gfCNCPoint5[26380] = {X 520.4681, Y 51.2791, Z -8.0000, A 0.000, B 0.000, C 0.000 }
gfCNCPoint5[26381] = {X 519.7998, Y 51.2791, Z -8.0000, A 0.000, B 0.000, C 0.000 }
gfCNCPoint5[26382] = {X 518.8207, Y 51.1688, Z -8.0000, A 0.000, B 0.000, C 0.000 }
gfCNCPoint5[26383] = {X 517.8907, Y 50.8434, Z -8.0000, A 0.000, B 0.000, C 0.000 }
gfCNCPoint5[26384] = {X 517.0564, Y 50.3192, Z -8.0000, A 0.000, B 0.000, C 0.000 }
gfCNCPoint5[26385] = {X 516.3597, Y 49.6225, Z -8.0000, A 0.000, B 0.000, C 0.000 }
gfCNCPoint5[26386] = {X 515.8355, Y 48.7882, Z -8.0000, A 0.000, B 0.000, C 0.000 }
gfCNCPoint5[26387] = {X 515.5101, Y 47.8582, Z -8.0000, A 0.000, B 0.000, C 0.000 }
gfCNCPoint5[26388] = {X 515.3998, Y 46.8791, Z -8.0000, A 0.000, B 0.000, C 0.000 }
gfCNCPoint5[26389] = {X 515.3998, Y 39.9011, Z -8.0000, A 0.000, B 0.000, C 0.000 }
gfCNCPoint5[26390] = {X 515.5101, Y 38.9220, Z -8.0000, A 0.000, B 0.000, C 0.000 }
gfCNCPoint5[26391] = {X 515.8355, Y 37.9920, Z -8.0000, A 0.000, B 0.000, C 0.000 }
gfCNCPoint5[26392] = {X 516.3597, Y 37.1577, Z -8.0000, A 0.000, B 0.000, C 0.000 }
gfCNCPoint5[26393] = {X 517.0564, Y 36.4610, Z -8.0000, A 0.000, B 0.000, C 0.000 }
gfCNCPoint5[26394] = {X 517.8907, Y 35.9368, Z -8.0000, A 0.000, B 0.000, C 0.000 }
gfCNCPoint5[26395] = {X 518.8207, Y 35.6114, Z -8.0000, A 0.000, B 0.000, C 0.000 }
gfCNCPoint5[26396] = {X 519.7998, Y 35.5011, Z -8.0000, A 0.000, B 0.000, C 0.000 }
gfCNCPoint5[26397] = {X 520.5280, Y 35.5015, Z -8.0000, A 0.000, B 0.000, C 0.000 }
gfCNCPoint5[26398] = {X 521.3612, Y 35.5927, Z -8.0000, A 0.000, B 0.000, C 0.000 }
gfCNCPoint5[26399] = {X 522.1620, Y 35.8402, Z -8.0000, A 0.000, B 0.000, C 0.000 }
gfCNCPoint5[26400] = {X 522.9013, Y 36.2351, Z -8.0000, A 0.000, B 0.000, C 0.000 }
gfCNCPoint5[26401] = {X 523.5524, Y 36.7630, Z -8.0000, A 0.000, B 0.000, C 0.000 }
gfCNCPoint5[26402] = {X 524.0915, Y 37.4048, Z -8.0000, A 0.000, B 0.000, C 0.000 }
gfCNCPoint5[26403] = {X 534.5519, Y 37.4048, Z -8.0000, A 0.000, B 0.000, C 0.000 }
gfCNCPoint5[26404] = {X 534.5519, Y 34.0464, Z -8.0000, A 0.000, B 0.000, C 0.000 }
gfCNCPoint5[26405] = {X 530.1514, Y 34.0463, Z -8.0000, A 0.000, B 0.000, C 0.000 }
gfCNCPoint5[26406] = {X 529.6037, Y 34.6963, Z -8.0000, A 0.000, B 0.000, C 0.000 }
gfCNCPoint5[26407] = {X 528.9413, Y 35.2289, Z -8.0000, A 0.000, B 0.000, C 0.000 }
gfCNCPoint5[26408] = {X 528.1888, Y 35.6242, Z -8.0000, A 0.000, B 0.000, C 0.000 }
gfCNCPoint5[26409] = {X 527.3744, Y 35.8674, Z -8.0000, A 0.000, B 0.000, C 0.000 }
gfCNCPoint5[26410] = {X 526.5283, Y 35.9495, Z -8.0000, A 0.000, B 0.000, C 0.000 }
gfCNCPoint5[26411] = {X 525.8868, Y 35.9495, Z -8.0000, A 0.000, B 0.000, C 0.000 }
gfCNCPoint5[26412] = {X 524.9077, Y 35.8391, Z -8.0000, A 0.000, B 0.000, C 0.000 }
gfCNCPoint5[26413] = {X 523.9777, Y 35.5137, Z -8.0000, A 0.000, B 0.000, C 0.000 }
gfCNCPoint5[26414] = {X 523.1434, Y 34.9895, Z -8.0000, A 0.000, B 0.000, C 0.000 }
gfCNCPoint5[26415] = {X 522.4467, Y 34.2928, Z -8.0000, A 0.000, B 0.000, C 0.000 }
gfCNCPoint5[26416] = {X 521.9225, Y 33.4585, Z -8.0000, A 0.000, B 0.000, C 0.000 }
gfCNCPoint5[26417] = {X 521.5971, Y 32.5285, Z -8.0000, A 0.000, B 0.000, C 0.000 }
gfCNCPoint5[26418] = {X 521.4868, Y 31.5495, Z -8.0000, A 0.000, B 0.000, C 0.000 }
gfCNCPoint5[26419] = {X 521.4868, Y 24.5714, Z -8.0000, A 0.000, B 0.000, C 0.000 }
gfCNCPoint5[26420] = {X 521.5971, Y 23.5923, Z -8.0000, A 0.000, B 0.000, C 0.000 }
gfCNCPoint5[26421] = {X 521.9225, Y 22.6623, Z -8.0000, A 0.000, B 0.000, C 0.000 }
gfCNCPoint5[26422] = {X 522.4467, Y 21.8281, Z -8.0000, A 0.000, B 0.000, C 0.000 }
gfCNCPoint5[26423] = {X 523.1434, Y 21.1314, Z -8.0000, A 0.000, B 0.000, C 0.000 }
gfCNCPoint5[26424] = {X 523.9777, Y 20.6072, Z -8.0000, A 0.000, B 0.000, C 0.000 }
gfCNCPoint5[26425] = {X 524.9077, Y 20.2817, Z -8.0000, A 0.000, B 0.000, C 0.000 }
gfCNCPoint5[26426] = {X 525.8868, Y 20.1714, Z -8.0000, A 0.000, B 0.000, C 0.000 }
gfCNCPoint5[26427] = {X 526.5702, Y 20.1716, Z -8.0000, A 0.000, B 0.000, C 0.000 }
gfCNCPoint5[26428] = {X 527.4020, Y 20.2590, Z -8.0000, A 0.000, B 0.000, C 0.000 }
gfCNCPoint5[26429] = {X 528.2022, Y 20.5022, Z -8.0000, A 0.000, B 0.000, C 0.000 }
gfCNCPoint5[26430] = {X 528.9419, Y 20.8924, Z -8.0000, A 0.000, B 0.000, C 0.000 }
gfCNCPoint5[26431] = {X 529.5945, Y 21.4156, Z -8.0000, A 0.000, B 0.000, C 0.000 }
gfCNCPoint5[26432] = {X 530.1362, Y 22.0527, Z -8.0000, A 0.000, B 0.000, C 0.000 }
gfCNCPoint5[26433] = {X 534.5519, Y 22.0527, Z -8.0000, A 0.000, B 0.000, C 0.000 }
gfCNCPoint5[26434] = {X 534.5519, Y 19.7828, Z -8.0000, A 0.000, B 0.000, C 0.000 }
gfCNCPoint5[26435] = {X 528.8197, Y 19.7828, Z -8.0000, A 0.000, B 0.000, C 0.000 }
gfCNCPoint5[26436] = {X 528.8197, Y 20.2628, Z -8.0000, A 0.000, B 0.000, C 0.000 }
gfCNCPoint5[26437] = {X 534.0719, Y 20.2628, Z -8.0000, A 0.000, B 0.000, C 0.000 }
gfCNCPoint5[26438] = {X 534.0719, Y 21.5727, Z -8.0000, A 0.000, B 0.000, C 0.000 }
gfCNCPoint5[26439] = {X 530.3784, Y 21.5727, Z -8.0000, A 0.000, B 0.000, C 0.000 }
gfCNCPoint5[26440] = {X 529.6681, Y 20.8356, Z -8.0000, A 0.000, B 0.000, C 0.000 }
gfCNCPoint5[26441] = {X 528.8197, Y 20.2628, Z -8.0000, A 0.000, B 0.000, C 0.000 }
gfCNCPoint5[26442] = {X 528.8197, Y 19.7828, Z -8.0000, A 0.000, B 0.000, C 0.000 }
gfCNCPoint5[26443] = {X 524.2336, Y 19.7828, Z -8.0000, A 0.000, B 0.000, C 0.000 }
gfCNCPoint5[26444] = {X 523.6859, Y 20.4327, Z -8.0000, A 0.000, B 0.000, C 0.000 }
gfCNCPoint5[26445] = {X 523.0235, Y 20.9652, Z -8.0000, A 0.000, B 0.000, C 0.000 }
gfCNCPoint5[26446] = {X 522.2711, Y 21.3604, Z -8.0000, A 0.000, B 0.000, C 0.000 }
gfCNCPoint5[26447] = {X 521.4567, Y 21.6036, Z -8.0000, A 0.000, B 0.000, C 0.000 }
gfCNCPoint5[26448] = {X 520.6107, Y 21.6857, Z -8.0000, A 0.000, B 0.000, C 0.000 }
gfCNCPoint5[26449] = {X 519.9691, Y 21.6857, Z -8.0000, A 0.000, B 0.000, C 0.000 }
gfCNCPoint5[26450] = {X 518.9900, Y 21.5754, Z -8.0000, A 0.000, B 0.000, C 0.000 }
gfCNCPoint5[26451] = {X 518.0600, Y 21.2500, Z -8.0000, A 0.000, B 0.000, C 0.000 }
gfCNCPoint5[26452] = {X 517.2257, Y 20.7258, Z -8.0000, A 0.000, B 0.000, C 0.000 }
gfCNCPoint5[26453] = {X 516.5290, Y 20.0291, Z -8.0000, A 0.000, B 0.000, C 0.000 }
gfCNCPoint5[26454] = {X 516.0048, Y 19.1948, Z -8.0000, A 0.000, B 0.000, C 0.000 }
gfCNCPoint5[26455] = {X 515.6794, Y 18.2648, Z -8.0000, A 0.000, B 0.000, C 0.000 }
gfCNCPoint5[26456] = {X 515.5691, Y 17.2857, Z -8.0000, A 0.000, B 0.000, C 0.000 }
gfCNCPoint5[26457] = {X 515.5691, Y 10.3077, Z -8.0000, A 0.000, B 0.000, C 0.000 }
gfCNCPoint5[26458] = {X 515.6394, Y 9.5244, Z -8.0000, A 0.000, B 0.000, C 0.000 }
gfCNCPoint5[26459] = {X 515.8480, Y 8.7661, Z -8.0000, A 0.000, B 0.000, C 0.000 }
gfCNCPoint5[26460] = {X 516.1883, Y 8.0570, Z -8.0000, A 0.000, B 0.000, C 0.000 }
gfCNCPoint5[26461] = {X 516.6494, Y 7.4199, Z -8.0000, A 0.000, B 0.000, C 0.000 }
gfCNCPoint5[26462] = {X 516.2873, Y 7.1048, Z -8.0000, A 0.000, B 0.000, C 0.000 }
gfCNCPoint5[26463] = {X 370.1008, Y 7.1048, Z -8.0000, A 0.000, B 0.000, C 0.000 }
gfCNCPoint5[26464] = {X 371.1247, Y 8.7921, Z -8.0000, A 0.000, B 0.000, C 0.000 }
gfCNCPoint5[26465] = {X 372.0360, Y 10.5428, Z -8.0000, A 0.000, B 0.000, C 0.000 }
gfCNCPoint5[26466] = {X 372.8329, Y 12.3542, Z -8.0000, A 0.000, B 0.000, C 0.000 }
gfCNCPoint5[26467] = {X 373.5091, Y 14.2140, Z -8.0000, A 0.000, B 0.000, C 0.000 }
gfCNCPoint5[26468] = {X 374.0619, Y 16.1141, Z -8.0000, A 0.000, B 0.000, C 0.000 }
gfCNCPoint5[26469] = {X 374.6092, Y 18.6904, Z -8.0000, A 0.000, B 0.000, C 0.000 }
gfCNCPoint5[26470] = {X 374.9714, Y 21.2992, Z -8.0000, A 0.000, B 0.000, C 0.000 }
gfCNCPoint5[26471] = {X 375.1469, Y 23.9271, Z -8.0000, A 0.000, B 0.000, C 0.000 }
gfCNCPoint5[26472] = {X 375.1347, Y 26.5608, Z -8.0000, A 0.000, B 0.000, C 0.000 }
gfCNCPoint5[26473] = {X 374.9349, Y 29.1870, Z -8.0000, A 0.000, B 0.000, C 0.000 }
gfCNCPoint5[26474] = {X 374.5485, Y 31.7923, Z -8.0000, A 0.000, B 0.000, C 0.000 }
gfCNCPoint5[26475] = {X 386.3483, Y 33.9749, Z -8.0000, A 0.000, B 0.000, C 0.000 }
gfCNCPoint5[26476] = {X 386.2676, Y 34.4005, Z -8.0000, A 0.000, B 0.000, C 0.000 }
gfCNCPoint5[26477] = {X 386.1832, Y 34.8254, Z -8.0000, A 0.000, B 0.000, C 0.000 }
gfCNCPoint5[26478] = {X 386.0243, Y 35.5742, Z -8.0000, A 0.000, B 0.000, C 0.000 }
gfCNCPoint5[26479] = {X 385.8518, Y 36.3200, Z -8.0000, A 0.000, B 0.000, C 0.000 }
gfCNCPoint5[26480] = {X 386.9552, Y 36.3200, Z -8.0000, A 0.000, B 0.000, C 0.000 }
gfCNCPoint5[26481] = {X 386.9552, Y 35.0303, Z -8.0000, A 0.000, B 0.000, C 0.000 }
gfCNCPoint5[26482] = {X 386.3483, Y 33.9749, Z -8.0000, A 0.000, B 0.000, C 0.000 }
gfCNCPoint5[26483] = {X 383.9884, Y 33.5384, Z -8.0000, A 0.000, B 0.000, C 0.000 }
gfCNCPoint5[26484] = {X 383.9116, Y 33.9435, Z -8.0000, A 0.000, B 0.000, C 0.000 }
gfCNCPoint5[26485] = {X 383.8312, Y 34.3479, Z -8.0000, A 0.000, B 0.000, C 0.000 }
gfCNCPoint5[26486] = {X 383.6813, Y 35.0543, Z -8.0000, A 0.000, B 0.000, C 0.000 }
gfCNCPoint5[26487] = {X 383.5186, Y 35.7577, Z -8.0000, A 0.000, B 0.000, C 0.000 }
gfCNCPoint5[26488] = {X 383.1288, Y 37.2470, Z -8.0000, A 0.000, B 0.000, C 0.000 }
gfCNCPoint5[26489] = {X 382.6813, Y 38.7200, Z -8.0000, A 0.000, B 0.000, C 0.000 }
gfCNCPoint5[26490] = {X 388.0597, Y 38.7200, Z -8.0000, A 0.000, B 0.000, C 0.000 }
gfCNCPoint5[26491] = {X 388.4821, Y 38.7246, Z -8.0000, A 0.000, B 0.000, C 0.000 }
gfCNCPoint5[26492] = {X 388.9043, Y 38.7385, Z -8.0000, A 0.000, B 0.000, C 0.000 }
gfCNCPoint5[26493] = {X 389.1204, Y 38.2363, Z -8.0000, A 0.000, B 0.000, C 0.000 }
gfCNCPoint5[26494] = {X 389.3552, Y 37.7427, Z -8.0000, A 0.000, B 0.000, C 0.000 }
gfCNCPoint5[26495] = {X 389.3552, Y 34.3894, Z -8.0000, A 0.000, B 0.000, C 0.000 }
gfCNCPoint5[26496] = {X 384.7465, Y 26.3749, Z -8.0000, A 0.000, B 0.000, C 0.000 }
gfCNCPoint5[26497] = {X 384.6173, Y 28.7747, Z -8.0000, A 0.000, B 0.000, C 0.000 }
gfCNCPoint5[26498] = {X 384.3643, Y 31.1647, Z -8.0000, A 0.000, B 0.000, C 0.000 }
gfCNCPoint5[26499] = {X 383.9884, Y 33.5384, Z -8.0000, A 0.000, B 0.000, C 0.000 }
gfCNCPoint5[26500] = {X 381.6284, Y 33.1019, Z -8.0000, A 0.000, B 0.000, C 0.000 }
gfCNCPoint5[26501] = {X 381.5555, Y 33.4865, Z -8.0000, A 0.000, B 0.000, C 0.000 }
gfCNCPoint5[26502] = {X 381.4792, Y 33.8705, Z -8.0000, A 0.000, B 0.000, C 0.000 }
gfCNCPoint5[26503] = {X 380.9979, Y 35.9396, Z -8.0000, A 0.000, B 0.000, C 0.000 }
gfCNCPoint5[26504] = {X 380.3990, Y 37.9777, Z -8.0000, A 0.000, B 0.000, C 0.000 }
gfCNCPoint5[26505] = {X 379.8437, Y 39.5622, Z -8.0000, A 0.000, B 0.000, C 0.000 }
gfCNCPoint5[26506] = {X 379.2173, Y 41.1200, Z -8.0000, A 0.000, B 0.000, C 0.000 }
gfCNCPoint5[26507] = {X 388.0597, Y 41.1200, Z -8.0000, A 0.000, B 0.000, C 0.000 }
gfCNCPoint5[26508] = {X 389.3256, Y 41.1675, Z -8.0000, A 0.000, B 0.000, C 0.000 }
gfCNCPoint5[26509] = {X 390.5844, Y 41.3099, Z -8.0000, A 0.000, B 0.000, C 0.000 }
gfCNCPoint5[26510] = {X 391.0709, Y 39.7838, Z -8.0000, A 0.000, B 0.000, C 0.000 }
gfCNCPoint5[26511] = {X 391.7552, Y 38.3355, Z -8.0000, A 0.000, B 0.000, C 0.000 }
gfCNCPoint5[26512] = {X 391.7552, Y 33.7486, Z -8.0000, A 0.000, B 0.000, C 0.000 }
gfCNCPoint5[26513] = {X 386.7075, Y 24.9707, Z -8.0000, A 0.000, B 0.000, C 0.000 }
gfCNCPoint5[26514] = {X 386.1105, Y 23.9508, Z -8.0000, A 0.000, B 0.000, C 0.000 }
gfCNCPoint5[26515] = {X 385.4975, Y 22.9404, Z -8.0000, A 0.000, B 0.000, C 0.000 }
gfCNCPoint5[26516] = {X 384.4699, Y 22.1514, Z -8.0000, A 0.000, B 0.000, C 0.000 }
gfCNCPoint5[26517] = {X 383.5327, Y 21.2569, Z -8.0000, A 0.000, B 0.000, C 0.000 }
gfCNCPoint5[26518] = {X 382.6966, Y 20.2672, Z -8.0000, A 0.000, B 0.000, C 0.000 }
gfCNCPoint5[26519] = {X 381.9714, Y 19.1936, Z -8.0000, A 0.000, B 0.000, C 0.000 }
gfCNCPoint5[26520] = {X 382.2245, Y 21.5571, Z -8.0000, A 0.000, B 0.000, C 0.000 }
gfCNCPoint5[26521] = {X 382.3499, Y 23.9308, Z -8.0000, A 0.000, B 0.000, C 0.000 }
gfCNCPoint5[26522] = {X 382.3474, Y 26.3077, Z -8.0000, A 0.000, B 0.000, C 0.000 }
gfCNCPoint5[26523] = {X 382.2249, Y 28.5838, Z -8.0000, A 0.000, B 0.000, C 0.000 }
gfCNCPoint5[26524] = {X 381.9850, Y 30.8506, Z -8.0000, A 0.000, B 0.000, C 0.000 }
gfCNCPoint5[26525] = {X 381.6284, Y 33.1019, Z -8.0000, A 0.000, B 0.000, C 0.000 }
gfCNCPoint5[26526] = {X 379.2684, Y 32.6654, Z -8.0000, A 0.000, B 0.000, C 0.000 }
gfCNCPoint5[26527] = {X 379.1994, Y 33.0295, Z -8.0000, A 0.000, B 0.000, C 0.000 }
gfCNCPoint5[26528] = {X 379.1271, Y 33.3931, Z -8.0000, A 0.000, B 0.000, C 0.000 }
gfCNCPoint5[26529] = {X 378.5771, Y 35.7000, Z -8.0000, A 0.000, B 0.000, C 0.000 }
gfCNCPoint5[26530] = {X 377.8708, Y 37.9640, Z -8.0000, A 0.000, B 0.000, C 0.000 }
gfCNCPoint5[26531] = {X 377.0114, Y 40.1744, Z -8.0000, A 0.000, B 0.000, C 0.000 }
gfCNCPoint5[26532] = {X 376.2302, Y 41.8694, Z -8.0000, A 0.000, B 0.000, C 0.000 }
gfCNCPoint5[26533] = {X 375.3590, Y 43.5200, Z -8.0000, A 0.000, B 0.000, C 0.000 }
gfCNCPoint5[26534] = {X 388.0597, Y 43.5200, Z -8.0000, A 0.000, B 0.000, C 0.000 }
gfCNCPoint5[26535] = {X 389.6072, Y 43.6029, Z -8.0000, A 0.000, B 0.000, C 0.000 }
gfCNCPoint5[26536] = {X 391.1370, Y 43.8508, Z -8.0000, A 0.000, B 0.000, C 0.000 }
gfCNCPoint5[26537] = {X 392.6316, Y 44.2607, Z -8.0000, A 0.000, B 0.000, C 0.000 }
gfCNCPoint5[26538] = {X 392.7236, Y 42.8756, Z -8.0000, A 0.000, B 0.000, C 0.000 }
gfCNCPoint5[26539] = {X 393.0129, Y 41.5179, Z -8.0000, A 0.000, B 0.000, C 0.000 }
gfCNCPoint5[26540] = {X 393.4934, Y 40.2155, Z -8.0000, A 0.000, B 0.000, C 0.000 }
gfCNCPoint5[26541] = {X 394.1552, Y 38.9952, Z -8.0000, A 0.000, B 0.000, C 0.000 }
gfCNCPoint5[26542] = {X 394.1552, Y 33.1077, Z -8.0000, A 0.000, B 0.000, C 0.000 }
gfCNCPoint5[26543] = {X 388.7881, Y 23.7743, Z -8.0000, A 0.000, B 0.000, C 0.000 }
gfCNCPoint5[26544] = {X 388.0333, Y 22.4902, Z -8.0000, A 0.000, B 0.000, C 0.000 }
gfCNCPoint5[26545] = {X 387.2543, Y 21.2208, Z -8.0000, A 0.000, B 0.000, C 0.000 }
gfCNCPoint5[26546] = {X 386.3070, Y 20.5563, Z -8.0000, A 0.000, B 0.000, C 0.000 }
gfCNCPoint5[26547] = {X 385.4458, Y 19.7835, Z -8.0000, A 0.000, B 0.000, C 0.000 }
gfCNCPoint5[26548] = {X 384.6829, Y 18.9135, Z -8.0000, A 0.000, B 0.000, C 0.000 }
gfCNCPoint5[26549] = {X 384.0293, Y 17.9587, Z -8.0000, A 0.000, B 0.000, C 0.000 }
gfCNCPoint5[26550] = {X 383.4406, Y 16.8105, Z -8.0000, A 0.000, B 0.000, C 0.000 }
gfCNCPoint5[26551] = {X 383.0098, Y 15.5941, Z -8.0000, A 0.000, B 0.000, C 0.000 }
gfCNCPoint5[26552] = {X 382.7447, Y 14.3312, Z -8.0000, A 0.000, B 0.000, C 0.000 }
gfCNCPoint5[26553] = {X 382.6498, Y 13.0443, Z -8.0000, A 0.000, B 0.000, C 0.000 }
gfCNCPoint5[26554] = {X 382.6496, Y 12.1868, Z -8.0000, A 0.000, B 0.000, C 0.000 }
gfCNCPoint5[26555] = {X 382.6507, Y 12.0458, Z -8.0000, A 0.000, B 0.000, C 0.000 }
gfCNCPoint5[26556] = {X 382.6537, Y 11.9048, Z -8.0000, A 0.000, B 0.000, C 0.000 }
gfCNCPoint5[26557] = {X 377.7930, Y 11.9048, Z -8.0000, A 0.000, B 0.000, C 0.000 }
gfCNCPoint5[26558] = {X 378.2878, Y 13.4079, Z -8.0000, A 0.000, B 0.000, C 0.000 }
gfCNCPoint5[26559] = {X 378.7141, Y 14.9319, Z -8.0000, A 0.000, B 0.000, C 0.000 }
gfCNCPoint5[26560] = {X 379.2175, Y 17.2103, Z -8.0000, A 0.000, B 0.000, C 0.000 }
gfCNCPoint5[26561] = {X 379.5928, Y 19.5133, Z -8.0000, A 0.000, B 0.000, C 0.000 }
gfCNCPoint5[26562] = {X 379.8616, Y 22.1413, Z -8.0000, A 0.000, B 0.000, C 0.000 }
gfCNCPoint5[26563] = {X 379.9637, Y 24.7812, Z -8.0000, A 0.000, B 0.000, C 0.000 }
gfCNCPoint5[26564] = {X 379.8985, Y 27.4221, Z -8.0000, A 0.000, B 0.000, C 0.000 }
gfCNCPoint5[26565] = {X 379.6665, Y 30.0537, Z -8.0000, A 0.000, B 0.000, C 0.000 }
gfCNCPoint5[26566] = {X 379.2684, Y 32.6654, Z -8.0000, A 0.000, B 0.000, C 0.000 }
gfCNCPoint5[26567] = {X 376.9085, Y 32.2288, Z -8.0000, A 0.000, B 0.000, C 0.000 }
gfCNCPoint5[26568] = {X 376.8433, Y 32.5725, Z -8.0000, A 0.000, B 0.000, C 0.000 }
gfCNCPoint5[26569] = {X 376.7751, Y 32.9156, Z -8.0000, A 0.000, B 0.000, C 0.000 }
gfCNCPoint5[26570] = {X 376.1777, Y 35.3682, Z -8.0000, A 0.000, B 0.000, C 0.000 }
gfCNCPoint5[26571] = {X 375.3905, Y 37.7667, Z -8.0000, A 0.000, B 0.000, C 0.000 }
gfCNCPoint5[26572] = {X 374.4185, Y 40.0964, Z -8.0000, A 0.000, B 0.000, C 0.000 }
gfCNCPoint5[26573] = {X 373.2674, Y 42.3430, Z -8.0000, A 0.000, B 0.000, C 0.000 }
gfCNCPoint5[26574] = {X 372.1530, Y 44.1780, Z -8.0000, A 0.000, B 0.000, C 0.000 }
gfCNCPoint5[26575] = {X 370.9191, Y 45.9349, Z -8.0000, A 0.000, B 0.000, C 0.000 }
gfCNCPoint5[26576] = {X 371.2191, Y 45.9237, Z -8.0000, A 0.000, B 0.000, C 0.000 }
gfCNCPoint5[26577] = {X 371.5193, Y 45.9200, Z -8.0000, A 0.000, B 0.000, C 0.000 }
gfCNCPoint5[26578] = {X 388.0597, Y 45.9200, Z -8.0000, A 0.000, B 0.000, C 0.000 }
gfCNCPoint5[26579] = {X 389.4143, Y 45.9962, Z -8.0000, A 0.000, B 0.000, C 0.000 }
gfCNCPoint5[26580] = {X 390.7519, Y 46.2238, Z -8.0000, A 0.000, B 0.000, C 0.000 }
gfCNCPoint5[26581] = {X 392.0555, Y 46.6000, Z -8.0000, A 0.000, B 0.000, C 0.000 }
gfCNCPoint5[26582] = {X 393.3087, Y 47.1200, Z -8.0000, A 0.000, B 0.000, C 0.000 }
gfCNCPoint5[26583] = {X 394.2237, Y 46.7243, Z -8.0000, A 0.000, B 0.000, C 0.000 }
gfCNCPoint5[26584] = {X 395.1681, Y 46.4053, Z -8.0000, A 0.000, B 0.000, C 0.000 }
gfCNCPoint5[26585] = {X 395.0678, Y 45.7292, Z -8.0000, A 0.000, B 0.000, C 0.000 }
gfCNCPoint5[26586] = {X 395.0314, Y 45.0468, Z -8.0000, A 0.000, B 0.000, C 0.000 }
gfCNCPoint5[26587] = {X 395.0316, Y 44.1296, Z -8.0000, A 0.000, B 0.000, C 0.000 }
gfCNCPoint5[26588] = {X 395.1397, Y 42.9564, Z -8.0000, A 0.000, B 0.000, C 0.000 }
gfCNCPoint5[26589] = {X 395.4356, Y 41.8161, Z -8.0000, A 0.000, B 0.000, C 0.000 }
gfCNCPoint5[26590] = {X 395.9116, Y 40.7384, Z -8.0000, A 0.000, B 0.000, C 0.000 }
gfCNCPoint5[26591] = {X 396.5552, Y 39.7516, Z -8.0000, A 0.000, B 0.000, C 0.000 }
gfCNCPoint5[26592] = {X 396.5552, Y 32.4669, Z -8.0000, A 0.000, B 0.000, C 0.000 }
gfCNCPoint5[26593] = {X 390.8686, Y 22.5779, Z -8.0000, A 0.000, B 0.000, C 0.000 }
gfCNCPoint5[26594] = {X 390.0503, Y 21.1873, Z -8.0000, A 0.000, B 0.000, C 0.000 }
gfCNCPoint5[26595] = {X 389.2044, Y 19.8133, Z -8.0000, A 0.000, B 0.000, C 0.000 }
gfCNCPoint5[26596] = {X 389.0604, Y 19.6016, Z -8.0000, A 0.000, B 0.000, C 0.000 }
gfCNCPoint5[26597] = {X 388.9019, Y 19.4005, Z -8.0000, A 0.000, B 0.000, C 0.000 }
gfCNCPoint5[26598] = {X 387.8143, Y 18.6886, Z -8.0000, A 0.000, B 0.000, C 0.000 }
gfCNCPoint5[26599] = {X 386.8707, Y 17.7945, Z -8.0000, A 0.000, B 0.000, C 0.000 }
gfCNCPoint5[26600] = {X 386.1011, Y 16.7469, Z -8.0000, A 0.000, B 0.000, C 0.000 }
gfCNCPoint5[26601] = {X 385.5302, Y 15.5791, Z -8.0000, A 0.000, B 0.000, C 0.000 }
gfCNCPoint5[26602] = {X 385.1760, Y 14.3284, Z -8.0000, A 0.000, B 0.000, C 0.000 }
gfCNCPoint5[26603] = {X 385.0498, Y 13.0347, Z -8.0000, A 0.000, B 0.000, C 0.000 }
gfCNCPoint5[26604] = {X 385.0496, Y 12.1868, Z -8.0000, A 0.000, B 0.000, C 0.000 }
gfCNCPoint5[26605] = {X 385.0504, Y 12.0808, Z -8.0000, A 0.000, B 0.000, C 0.000 }
gfCNCPoint5[26606] = {X 385.0527, Y 11.9747, Z -8.0000, A 0.000, B 0.000, C 0.000 }
gfCNCPoint5[26607] = {X 385.1994, Y 10.7176, Z -8.0000, A 0.000, B 0.000, C 0.000 }
gfCNCPoint5[26608] = {X 385.5617, Y 9.5048, Z -8.0000, A 0.000, B 0.000, C 0.000 }
gfCNCPoint5[26609] = {X 374.2000, Y 9.5048, Z -8.0000, A 0.000, B 0.000, C 0.000 }
gfCNCPoint5[26610] = {X 374.9081, Y 11.0880, Z -8.0000, A 0.000, B 0.000, C 0.000 }
gfCNCPoint5[26611] = {X 375.5309, Y 12.7067, Z -8.0000, A 0.000, B 0.000, C 0.000 }
gfCNCPoint5[26612] = {X 375.9918, Y 14.1066, Z -8.0000, A 0.000, B 0.000, C 0.000 }
gfCNCPoint5[26613] = {X 376.3888, Y 15.5259, Z -8.0000, A 0.000, B 0.000, C 0.000 }
gfCNCPoint5[26614] = {X 376.9722, Y 18.2705, Z -8.0000, A 0.000, B 0.000, C 0.000 }
gfCNCPoint5[26615] = {X 377.3585, Y 21.0497, Z -8.0000, A 0.000, B 0.000, C 0.000 }
gfCNCPoint5[26616] = {X 377.5457, Y 23.8494, Z -8.0000, A 0.000, B 0.000, C 0.000 }
gfCNCPoint5[26617] = {X 377.5329, Y 26.6554, Z -8.0000, A 0.000, B 0.000, C 0.000 }
gfCNCPoint5[26618] = {X 377.3201, Y 29.4532, Z -8.0000, A 0.000, B 0.000, C 0.000 }
gfCNCPoint5[26619] = {X 376.9085, Y 32.2288, Z -8.0000, A 0.000, B 0.000, C 0.000 }
gfCNCPoint5[26620] = {X 374.5485, Y 31.7923, Z -8.0000, A 0.000, B 0.000, C 0.000 }
gfCNCPoint5[26621] = {X 374.4872, Y 32.1155, Z -8.0000, A 0.000, B 0.000, C 0.000 }
gfCNCPoint5[26622] = {X 374.4231, Y 32.4381, Z -8.0000, A 0.000, B 0.000, C 0.000 }
gfCNCPoint5[26623] = {X 373.8982, Y 34.6095, Z -8.0000, A 0.000, B 0.000, C 0.000 }
gfCNCPoint5[26624] = {X 373.2127, Y 36.7356, Z -8.0000, A 0.000, B 0.000, C 0.000 }
gfCNCPoint5[26625] = {X 372.3703, Y 38.8046, Z -8.0000, A 0.000, B 0.000, C 0.000 }
gfCNCPoint5[26626] = {X 371.3758, Y 40.8049, Z -8.0000, A 0.000, B 0.000, C 0.000 }
gfCNCPoint5[26627] = {X 370.2347, Y 42.7254, Z -8.0000, A 0.000, B 0.000, C 0.000 }
gfCNCPoint5[26628] = {X 368.9534, Y 44.5554, Z -8.0000, A 0.000, B 0.000, C 0.000 }
gfCNCPoint5[26629] = {X 367.5572, Y 46.2628, Z -8.0000, A 0.000, B 0.000, C 0.000 }
gfCNCPoint5[26630] = {X 366.0280, Y 47.8522, Z -8.0000, A 0.000, B 0.000, C 0.000 }
gfCNCPoint5[26631] = {X 364.3756, Y 49.3132, Z -8.0000, A 0.000, B 0.000, C 0.000 }
gfCNCPoint5[26632] = {X 362.6108, Y 50.6362, Z -8.0000, A 0.000, B 0.000, C 0.000 }
gfCNCPoint5[26633] = {X 360.7452, Y 51.8127, Z -8.0000, A 0.000, B 0.000, C 0.000 }
gfCNCPoint5[26634] = {X 358.7908, Y 52.8350, Z -8.0000, A 0.000, B 0.000, C 0.000 }
gfCNCPoint5[26635] = {X 358.6057, Y 52.9216, Z -8.0000, A 0.000, B 0.000, C 0.000 }
gfCNCPoint5[26636] = {X 358.4200, Y 53.0069, Z -8.0000, A 0.000, B 0.000, C 0.000 }
gfCNCPoint5[26637] = {X 356.1467, Y 53.8835, Z -8.0000, A 0.000, B 0.000, C 0.000 }
gfCNCPoint5[26638] = {X 353.8065, Y 54.5619, Z -8.0000, A 0.000, B 0.000, C 0.000 }
gfCNCPoint5[26639] = {X 351.4168, Y 55.0371, Z -8.0000, A 0.000, B 0.000, C 0.000 }
gfCNCPoint5[26640] = {X 348.9952, Y 55.3056, Z -8.0000, A 0.000, B 0.000, C 0.000 }
gfCNCPoint5[26641] = {X 349.9664, Y 69.6728, Z -8.0000, A 0.000, B 0.000, C 0.000 }
gfCNCPoint5[26642] = {X 348.6648, Y 69.7409, Z -8.0000, A 0.000, B 0.000, C 0.000 }
gfCNCPoint5[26643] = {X 347.3618, Y 69.7693, Z -8.0000, A 0.000, B 0.000, C 0.000 }
gfCNCPoint5[26644] = {X 346.5844, Y 69.7785, Z -8.0000, A 0.000, B 0.000, C 0.000 }
gfCNCPoint5[26645] = {X 345.8070, Y 69.7737, Z -8.0000, A 0.000, B 0.000, C 0.000 }
gfCNCPoint5[26646] = {X 345.5918, Y 70.1904, Z -8.0000, A 0.000, B 0.000, C 0.000 }
gfCNCPoint5[26647] = {X 345.3684, Y 70.6028, Z -8.0000, A 0.000, B 0.000, C 0.000 }
gfCNCPoint5[26648] = {X 347.2082, Y 70.6201, Z -8.0000, A 0.000, B 0.000, C 0.000 }
gfCNCPoint5[26649] = {X 349.0480, Y 70.6084, Z -8.0000, A 0.000, B 0.000, C 0.000 }
gfCNCPoint5[26650] = {X 349.7516, Y 70.6081, Z -8.0000, A 0.000, B 0.000, C 0.000 }
gfCNCPoint5[26651] = {X 350.4553, Y 70.6025, Z -8.0000, A 0.000, B 0.000, C 0.000 }
gfCNCPoint5[26652] = {X 350.2058, Y 70.1403, Z -8.0000, A 0.000, B 0.000, C 0.000 }
gfCNCPoint5[26653] = {X 349.9664, Y 69.6728, Z -8.0000, A 0.000, B 0.000, C 0.000 }
gfCNCPoint5[26654] = {X 349.8045, Y 67.2783, Z -8.0000, A 0.000, B 0.000, C 0.000 }
gfCNCPoint5[26655] = {X 348.5675, Y 67.3429, Z -8.0000, A 0.000, B 0.000, C 0.000 }
gfCNCPoint5[26656] = {X 347.3291, Y 67.3695, Z -8.0000, A 0.000, B 0.000, C 0.000 }
gfCNCPoint5[26657] = {X 345.8126, Y 67.3735, Z -8.0000, A 0.000, B 0.000, C 0.000 }
gfCNCPoint5[26658] = {X 344.2969, Y 67.3217, Z -8.0000, A 0.000, B 0.000, C 0.000 }
gfCNCPoint5[26659] = {X 343.8118, Y 68.3945, Z -8.0000, A 0.000, B 0.000, C 0.000 }
gfCNCPoint5[26660] = {X 343.2692, Y 69.4395, Z -8.0000, A 0.000, B 0.000, C 0.000 }
gfCNCPoint5[26661] = {X 342.7891, Y 70.2628, Z -8.0000, A 0.000, B 0.000, C 0.000 }
gfCNCPoint5[26662] = {X 342.2734, Y 71.0641, Z -8.0000, A 0.000, B 0.000, C 0.000 }
gfCNCPoint5[26663] = {X 342.2736, Y 72.9104, Z -8.0000, A 0.000, B 0.000, C 0.000 }
gfCNCPoint5[26664] = {X 343.8000, Y 72.9662, Z -8.0000, A 0.000, B 0.000, C 0.000 }
gfCNCPoint5[26665] = {X 345.3269, Y 73.0024, Z -8.0000, A 0.000, B 0.000, C 0.000 }
gfCNCPoint5[26666] = {X 347.1940, Y 73.0201, Z -8.0000, A 0.000, B 0.000, C 0.000 }
gfCNCPoint5[26667] = {X 349.0612, Y 73.0085, Z -8.0000, A 0.000, B 0.000, C 0.000 }
gfCNCPoint5[26668] = {X 349.7722, Y 73.0080, Z -8.0000, A 0.000, B 0.000, C 0.000 }
gfCNCPoint5[26669] = {X 350.4831, Y 73.0024, Z -8.0000, A 0.000, B 0.000, C 0.000 }
gfCNCPoint5[26670] = {X 352.0210, Y 72.9723, Z -8.0000, A 0.000, B 0.000, C 0.000 }
gfCNCPoint5[26671] = {X 353.5582, Y 72.9179, Z -8.0000, A 0.000, B 0.000, C 0.000 }
gfCNCPoint5[26672] = {X 353.5581, Y 71.0756, Z -8.0000, A 0.000, B 0.000, C 0.000 }
gfCNCPoint5[26673] = {X 353.0382, Y 70.2687, Z -8.0000, A 0.000, B 0.000, C 0.000 }
gfCNCPoint5[26674] = {X 352.5547, Y 69.4396, Z -8.0000, A 0.000, B 0.000, C 0.000 }
gfCNCPoint5[26675] = {X 351.9680, Y 68.3027, Z -8.0000, A 0.000, B 0.000, C 0.000 }
gfCNCPoint5[26676] = {X 351.4495, Y 67.1332, Z -8.0000, A 0.000, B 0.000, C 0.000 }
gfCNCPoint5[26677] = {X 350.6278, Y 67.2142, Z -8.0000, A 0.000, B 0.000, C 0.000 }
gfCNCPoint5[26678] = {X 349.8045, Y 67.2783, Z -8.0000, A 0.000, B 0.000, C 0.000 }
gfCNCPoint5[26679] = {X 349.6427, Y 64.8838, Z -8.0000, A 0.000, B 0.000, C 0.000 }
gfCNCPoint5[26680] = {X 348.4702, Y 64.9448, Z -8.0000, A 0.000, B 0.000, C 0.000 }
gfCNCPoint5[26681] = {X 347.2964, Y 64.9696, Z -8.0000, A 0.000, B 0.000, C 0.000 }
gfCNCPoint5[26682] = {X 344.9826, Y 64.9504, Z -8.0000, A 0.000, B 0.000, C 0.000 }
gfCNCPoint5[26683] = {X 342.6741, Y 64.7932, Z -8.0000, A 0.000, B 0.000, C 0.000 }
gfCNCPoint5[26684] = {X 341.9396, Y 66.7276, Z -8.0000, A 0.000, B 0.000, C 0.000 }
gfCNCPoint5[26685] = {X 341.0024, Y 68.5724, Z -8.0000, A 0.000, B 0.000, C 0.000 }
gfCNCPoint5[26686] = {X 339.8733, Y 70.3064, Z -8.0000, A 0.000, B 0.000, C 0.000 }
gfCNCPoint5[26687] = {X 339.8738, Y 75.1877, Z -8.0000, A 0.000, B 0.000, C 0.000 }
gfCNCPoint5[26688] = {X 344.4720, Y 75.3853, Z -8.0000, A 0.000, B 0.000, C 0.000 }
gfCNCPoint5[26689] = {X 349.0745, Y 75.4085, Z -8.0000, A 0.000, B 0.000, C 0.000 }
gfCNCPoint5[26690] = {X 352.5183, Y 75.3586, Z -8.0000, A 0.000, B 0.000, C 0.000 }
gfCNCPoint5[26691] = {X 355.9583, Y 75.1895, Z -8.0000, A 0.000, B 0.000, C 0.000 }
gfCNCPoint5[26692] = {X 355.9580, Y 70.3167, Z -8.0000, A 0.000, B 0.000, C 0.000 }
gfCNCPoint5[26693] = {X 355.0507, Y 68.9593, Z -8.0000, A 0.000, B 0.000, C 0.000 }
gfCNCPoint5[26694] = {X 354.2615, Y 67.5299, Z -8.0000, A 0.000, B 0.000, C 0.000 }
gfCNCPoint5[26695] = {X 353.5961, Y 66.0388, Z -8.0000, A 0.000, B 0.000, C 0.000 }
gfCNCPoint5[26696] = {X 353.0592, Y 64.4968, Z -8.0000, A 0.000, B 0.000, C 0.000 }
gfCNCPoint5[26697] = {X 351.3553, Y 64.7290, Z -8.0000, A 0.000, B 0.000, C 0.000 }
gfCNCPoint5[26698] = {X 349.6427, Y 64.8838, Z -8.0000, A 0.000, B 0.000, C 0.000 }
gfCNCPoint5[26699] = {X 349.4808, Y 62.4892, Z -8.0000, A 0.000, B 0.000, C 0.000 }
gfCNCPoint5[26700] = {X 348.3729, Y 62.5468, Z -8.0000, A 0.000, B 0.000, C 0.000 }
gfCNCPoint5[26701] = {X 347.2638, Y 62.5698, Z -8.0000, A 0.000, B 0.000, C 0.000 }
gfCNCPoint5[26702] = {X 345.1284, Y 62.5542, Z -8.0000, A 0.000, B 0.000, C 0.000 }
gfCNCPoint5[26703] = {X 342.9976, Y 62.4133, Z -8.0000, A 0.000, B 0.000, C 0.000 }
gfCNCPoint5[26704] = {X 340.8787, Y 62.1476, Z -8.0000, A 0.000, B 0.000, C 0.000 }
gfCNCPoint5[26705] = {X 340.4890, Y 63.7352, Z -8.0000, A 0.000, B 0.000, C 0.000 }
gfCNCPoint5[26706] = {X 339.9479, Y 65.2779, Z -8.0000, A 0.000, B 0.000, C 0.000 }
gfCNCPoint5[26707] = {X 339.2604, Y 66.7611, Z -8.0000, A 0.000, B 0.000, C 0.000 }
gfCNCPoint5[26708] = {X 338.4329, Y 68.1710, Z -8.0000, A 0.000, B 0.000, C 0.000 }
gfCNCPoint5[26709] = {X 337.4732, Y 69.4944, Z -8.0000, A 0.000, B 0.000, C 0.000 }
gfCNCPoint5[26710] = {X 337.4740, Y 77.4231, Z -8.0000, A 0.000, B 0.000, C 0.000 }
gfCNCPoint5[26711] = {X 341.3406, Y 77.6726, Z -8.0000, A 0.000, B 0.000, C 0.000 }
gfCNCPoint5[26712] = {X 345.2131, Y 77.8012, Z -8.0000, A 0.000, B 0.000, C 0.000 }
gfCNCPoint5[26713] = {X 349.0878, Y 77.8086, Z -8.0000, A 0.000, B 0.000, C 0.000 }
gfCNCPoint5[26714] = {X 353.7276, Y 77.7150, Z -8.0000, A 0.000, B 0.000, C 0.000 }
gfCNCPoint5[26715] = {X 358.3584, Y 77.4101, Z -8.0000, A 0.000, B 0.000, C 0.000 }
gfCNCPoint5[26716] = {X 358.3580, Y 69.5036, Z -8.0000, A 0.000, B 0.000, C 0.000 }
gfCNCPoint5[26717] = {X 357.3473, Y 68.1041, Z -8.0000, A 0.000, B 0.000, C 0.000 }
gfCNCPoint5[26718] = {X 356.4848, Y 66.6087, Z -8.0000, A 0.000, B 0.000, C 0.000 }
gfCNCPoint5[26719] = {X 355.7796, Y 65.0331, Z -8.0000, A 0.000, B 0.000, C 0.000 }
gfCNCPoint5[26720] = {X 355.2390, Y 63.3936, Z -8.0000, A 0.000, B 0.000, C 0.000 }
gfCNCPoint5[26721] = {X 354.8687, Y 61.7076, Z -8.0000, A 0.000, B 0.000, C 0.000 }
gfCNCPoint5[26722] = {X 352.1897, Y 62.2016, Z -8.0000, A 0.000, B 0.000, C 0.000 }
gfCNCPoint5[26723] = {X 349.4808, Y 62.4892, Z -8.0000, A 0.000, B 0.000, C 0.000 }
gfCNCPoint5[26724] = {X 349.3189, Y 60.0947, Z -8.0000, A 0.000, B 0.000, C 0.000 }
gfCNCPoint5[26725] = {X 348.2756, Y 60.1487, Z -8.0000, A 0.000, B 0.000, C 0.000 }
gfCNCPoint5[26726] = {X 347.2311, Y 60.1699, Z -8.0000, A 0.000, B 0.000, C 0.000 }
gfCNCPoint5[26727] = {X 344.3950, Y 60.1157, Z -8.0000, A 0.000, B 0.000, C 0.000 }
gfCNCPoint5[26728] = {X 341.5732, Y 59.8251, Z -8.0000, A 0.000, B 0.000, C 0.000 }
gfCNCPoint5[26729] = {X 338.7856, Y 59.3000, Z -8.0000, A 0.000, B 0.000, C 0.000 }
gfCNCPoint5[26730] = {X 338.6401, Y 60.9992, Z -8.0000, A 0.000, B 0.000, C 0.000 }
gfCNCPoint5[26731] = {X 338.2964, Y 62.6696, Z -8.0000, A 0.000, B 0.000, C 0.000 }
gfCNCPoint5[26732] = {X 337.7591, Y 64.2881, Z -8.0000, A 0.000, B 0.000, C 0.000 }
gfCNCPoint5[26733] = {X 337.0358, Y 65.8325, Z -8.0000, A 0.000, B 0.000, C 0.000 }
gfCNCPoint5[26734] = {X 336.1363, Y 67.2813, Z -8.0000, A 0.000, B 0.000, C 0.000 }
gfCNCPoint5[26735] = {X 335.0731, Y 68.6147, Z -8.0000, A 0.000, B 0.000, C 0.000 }
gfCNCPoint5[26736] = {X 335.0742, Y 79.5851, Z -8.0000, A 0.000, B 0.000, C 0.000 }
gfCNCPoint5[26737] = {X 335.9841, Y 79.6946, Z -8.0000, A 0.000, B 0.000, C 0.000 }
gfCNCPoint5[26738] = {X 336.8962, Y 79.7838, Z -8.0000, A 0.000, B 0.000, C 0.000 }
gfCNCPoint5[26739] = {X 340.9592, Y 80.0566, Z -8.0000, A 0.000, B 0.000, C 0.000 }
gfCNCPoint5[26740] = {X 345.0290, Y 80.1982, Z -8.0000, A 0.000, B 0.000, C 0.000 }
gfCNCPoint5[26741] = {X 349.1011, Y 80.2086, Z -8.0000, A 0.000, B 0.000, C 0.000 }
gfCNCPoint5[26742] = {X 352.9063, Y 80.1484, Z -8.0000, A 0.000, B 0.000, C 0.000 }
gfCNCPoint5[26743] = {X 356.7068, Y 79.9494, Z -8.0000, A 0.000, B 0.000, C 0.000 }
gfCNCPoint5[26744] = {X 360.4975, Y 79.6116, Z -8.0000, A 0.000, B 0.000, C 0.000 }
gfCNCPoint5[26745] = {X 360.7585, Y 79.5816, Z -8.0000, A 0.000, B 0.000, C 0.000 }
gfCNCPoint5[26746] = {X 360.7579, Y 68.6224, Z -8.0000, A 0.000, B 0.000, C 0.000 }
gfCNCPoint5[26747] = {X 359.7292, Y 67.3403, Z -8.0000, A 0.000, B 0.000, C 0.000 }
gfCNCPoint5[26748] = {X 358.8524, Y 65.9498, Z -8.0000, A 0.000, B 0.000, C 0.000 }
gfCNCPoint5[26749] = {X 358.1389, Y 64.4689, Z -8.0000, A 0.000, B 0.000, C 0.000 }
gfCNCPoint5[26750] = {X 357.5978, Y 62.9167, Z -8.0000, A 0.000, B 0.000, C 0.000 }
gfCNCPoint5[26751] = {X 357.2361, Y 61.3132, Z -8.0000, A 0.000, B 0.000, C 0.000 }
gfCNCPoint5[26752] = {X 357.0916, Y 60.1642, Z -8.0000, A 0.000, B 0.000, C 0.000 }
gfCNCPoint5[26753] = {X 357.0395, Y 59.0073, Z -8.0000, A 0.000, B 0.000, C 0.000 }
gfCNCPoint5[26754] = {X 357.0394, Y 58.6407, Z -8.0000, A 0.000, B 0.000, C 0.000 }
gfCNCPoint5[26755] = {X 355.6990, Y 59.0316, Z -8.0000, A 0.000, B 0.000, C 0.000 }
gfCNCPoint5[26756] = {X 354.3434, Y 59.3657, Z -8.0000, A 0.000, B 0.000, C 0.000 }
gfCNCPoint5[26757] = {X 351.8451, Y 59.8264, Z -8.0000, A 0.000, B 0.000, C 0.000 }
gfCNCPoint5[26758] = {X 349.3189, Y 60.0947, Z -8.0000, A 0.000, B 0.000, C 0.000 }
gfCNCPoint5[26759] = {X 349.1570, Y 57.7002, Z -8.0000, A 0.000, B 0.000, C 0.000 }
gfCNCPoint5[26760] = {X 348.1783, Y 57.7507, Z -8.0000, A 0.000, B 0.000, C 0.000 }
gfCNCPoint5[26761] = {X 347.1985, Y 57.7700, Z -8.0000, A 0.000, B 0.000, C 0.000 }
gfCNCPoint5[26762] = {X 344.5555, Y 57.7210, Z -8.0000, A 0.000, B 0.000, C 0.000 }
gfCNCPoint5[26763] = {X 341.9258, Y 57.4511, Z -8.0000, A 0.000, B 0.000, C 0.000 }
gfCNCPoint5[26764] = {X 339.3279, Y 56.9621, Z -8.0000, A 0.000, B 0.000, C 0.000 }
gfCNCPoint5[26765] = {X 337.7710, Y 56.5589, Z -8.0000, A 0.000, B 0.000, C 0.000 }
gfCNCPoint5[26766] = {X 336.2366, Y 56.0770, Z -8.0000, A 0.000, B 0.000, C 0.000 }
gfCNCPoint5[26767] = {X 336.3521, Y 57.0354, Z -8.0000, A 0.000, B 0.000, C 0.000 }
gfCNCPoint5[26768] = {X 336.3907, Y 58.0000, Z -8.0000, A 0.000, B 0.000, C 0.000 }
gfCNCPoint5[26769] = {X 336.3907, Y 58.9560, Z -8.0000, A 0.000, B 0.000, C 0.000 }
gfCNCPoint5[26770] = {X 336.3894, Y 59.0961, Z -8.0000, A 0.000, B 0.000, C 0.000 }
gfCNCPoint5[26771] = {X 336.3864, Y 59.2361, Z -8.0000, A 0.000, B 0.000, C 0.000 }
gfCNCPoint5[26772] = {X 336.2429, Y 60.8001, Z -8.0000, A 0.000, B 0.000, C 0.000 }
gfCNCPoint5[26773] = {X 335.8983, Y 62.3325, Z -8.0000, A 0.000, B 0.000, C 0.000 }
gfCNCPoint5[26774] = {X 335.3584, Y 63.8074, Z -8.0000, A 0.000, B 0.000, C 0.000 }
gfCNCPoint5[26775] = {X 334.6323, Y 65.2000, Z -8.0000, A 0.000, B 0.000, C 0.000 }
gfCNCPoint5[26776] = {X 333.7321, Y 66.4871, Z -8.0000, A 0.000, B 0.000, C 0.000 }
gfCNCPoint5[26777] = {X 332.6730, Y 67.6468, Z -8.0000, A 0.000, B 0.000, C 0.000 }
gfCNCPoint5[26778] = {X 332.6744, Y 81.6385, Z -8.0000, A 0.000, B 0.000, C 0.000 }
gfCNCPoint5[26779] = {X 334.6775, Y 81.9535, Z -8.0000, A 0.000, B 0.000, C 0.000 }
gfCNCPoint5[26780] = {X 336.6930, Y 82.1752, Z -8.0000, A 0.000, B 0.000, C 0.000 }
gfCNCPoint5[26781] = {X 340.8281, Y 82.4530, Z -8.0000, A 0.000, B 0.000, C 0.000 }
gfCNCPoint5[26782] = {X 344.9701, Y 82.5976, Z -8.0000, A 0.000, B 0.000, C 0.000 }
gfCNCPoint5[26783] = {X 349.1145, Y 82.6086, Z -8.0000, A 0.000, B 0.000, C 0.000 }
gfCNCPoint5[26784] = {X 353.0020, Y 82.5466, Z -8.0000, A 0.000, B 0.000, C 0.000 }
gfCNCPoint5[26785] = {X 356.8846, Y 82.3428, Z -8.0000, A 0.000, B 0.000, C 0.000 }
gfCNCPoint5[26786] = {X 360.7571, Y 81.9975, Z -8.0000, A 0.000, B 0.000, C 0.000 }
gfCNCPoint5[26787] = {X 361.9615, Y 81.8404, Z -8.0000, A 0.000, B 0.000, C 0.000 }
gfCNCPoint5[26788] = {X 363.1586, Y 81.6348, Z -8.0000, A 0.000, B 0.000, C 0.000 }
gfCNCPoint5[26789] = {X 363.1579, Y 67.6526, Z -8.0000, A 0.000, B 0.000, C 0.000 }
gfCNCPoint5[26790] = {X 362.0720, Y 66.4624, Z -8.0000, A 0.000, B 0.000, C 0.000 }
gfCNCPoint5[26791] = {X 361.1542, Y 65.1383, Z -8.0000, A 0.000, B 0.000, C 0.000 }
gfCNCPoint5[26792] = {X 360.4208, Y 63.7038, Z -8.0000, A 0.000, B 0.000, C 0.000 }
gfCNCPoint5[26793] = {X 359.8848, Y 62.1845, Z -8.0000, A 0.000, B 0.000, C 0.000 }
gfCNCPoint5[26794] = {X 359.5557, Y 60.6074, Z -8.0000, A 0.000, B 0.000, C 0.000 }
gfCNCPoint5[26795] = {X 359.4395, Y 59.0005, Z -8.0000, A 0.000, B 0.000, C 0.000 }
gfCNCPoint5[26796] = {X 359.4393, Y 58.0000, Z -8.0000, A 0.000, B 0.000, C 0.000 }
gfCNCPoint5[26797] = {X 359.5340, Y 56.4906, Z -8.0000, A 0.000, B 0.000, C 0.000 }
gfCNCPoint5[26798] = {X 359.8165, Y 55.0048, Z -8.0000, A 0.000, B 0.000, C 0.000 }
gfCNCPoint5[26799] = {X 359.6067, Y 55.1030, Z -8.0000, A 0.000, B 0.000, C 0.000 }
gfCNCPoint5[26800] = {X 359.3960, Y 55.1995, Z -8.0000, A 0.000, B 0.000, C 0.000 }
gfCNCPoint5[26801] = {X 357.8730, Y 55.8165, Z -8.0000, A 0.000, B 0.000, C 0.000 }
gfCNCPoint5[26802] = {X 356.3192, Y 56.3513, Z -8.0000, A 0.000, B 0.000, C 0.000 }
gfCNCPoint5[26803] = {X 353.9699, Y 56.9895, Z -8.0000, A 0.000, B 0.000, C 0.000 }
gfCNCPoint5[26804] = {X 351.5775, Y 57.4400, Z -8.0000, A 0.000, B 0.000, C 0.000 }
gfCNCPoint5[26805] = {X 349.1570, Y 57.7002, Z -8.0000, A 0.000, B 0.000, C 0.000 }
gfCNCPoint5[26806] = {X 348.9952, Y 55.3056, Z -8.0000, A 0.000, B 0.000, C 0.000 }
gfCNCPoint5[26807] = {X 348.0811, Y 55.3526, Z -8.0000, A 0.000, B 0.000, C 0.000 }
gfCNCPoint5[26808] = {X 347.1659, Y 55.3701, Z -8.0000, A 0.000, B 0.000, C 0.000 }
gfCNCPoint5[26809] = {X 344.5859, Y 55.3183, Z -8.0000, A 0.000, B 0.000, C 0.000 }
gfCNCPoint5[26810] = {X 342.0206, Y 55.0386, Z -8.0000, A 0.000, B 0.000, C 0.000 }
gfCNCPoint5[26811] = {X 339.4900, Y 54.5333, Z -8.0000, A 0.000, B 0.000, C 0.000 }
gfCNCPoint5[26812] = {X 337.0139, Y 53.8063, Z -8.0000, A 0.000, B 0.000, C 0.000 }
gfCNCPoint5[26813] = {X 334.7573, Y 52.9276, Z -8.0000, A 0.000, B 0.000, C 0.000 }
gfCNCPoint5[26814] = {X 332.5814, Y 51.8647, Z -8.0000, A 0.000, B 0.000, C 0.000 }
gfCNCPoint5[26815] = {X 331.5882, Y 51.2806, Z -8.0000, A 0.000, B 0.000, C 0.000 }
gfCNCPoint5[26816] = {X 330.6189, Y 50.6578, Z -8.0000, A 0.000, B 0.000, C 0.000 }
gfCNCPoint5[26817] = {X 331.5832, Y 51.6115, Z -8.0000, A 0.000, B 0.000, C 0.000 }
gfCNCPoint5[26818] = {X 332.4047, Y 52.6907, Z -8.0000, A 0.000, B 0.000, C 0.000 }
gfCNCPoint5[26819] = {X 333.0673, Y 53.8741, Z -8.0000, A 0.000, B 0.000, C 0.000 }
gfCNCPoint5[26820] = {X 333.5581, Y 55.1385, Z -8.0000, A 0.000, B 0.000, C 0.000 }
gfCNCPoint5[26821] = {X 333.8672, Y 56.4590, Z -8.0000, A 0.000, B 0.000, C 0.000 }
gfCNCPoint5[26822] = {X 333.9598, Y 57.2270, Z -8.0000, A 0.000, B 0.000, C 0.000 }
gfCNCPoint5[26823] = {X 333.9907, Y 58.0000, Z -8.0000, A 0.000, B 0.000, C 0.000 }
gfCNCPoint5[26824] = {X 333.9907, Y 58.9476, Z -8.0000, A 0.000, B 0.000, C 0.000 }
gfCNCPoint5[26825] = {X 333.8760, Y 60.4022, Z -8.0000, A 0.000, B 0.000, C 0.000 }
gfCNCPoint5[26826] = {X 333.5448, Y 61.8233, Z -8.0000, A 0.000, B 0.000, C 0.000 }
gfCNCPoint5[26827] = {X 333.0045, Y 63.1788, Z -8.0000, A 0.000, B 0.000, C 0.000 }
gfCNCPoint5[26828] = {X 332.2673, Y 64.4381, Z -8.0000, A 0.000, B 0.000, C 0.000 }
gfCNCPoint5[26829] = {X 331.3499, Y 65.5728, Z -8.0000, A 0.000, B 0.000, C 0.000 }
gfCNCPoint5[26830] = {X 330.2729, Y 66.5573, Z -8.0000, A 0.000, B 0.000, C 0.000 }
gfCNCPoint5[26831] = {X 330.2746, Y 83.2031, Z -8.0000, A 0.000, B 0.000, C 0.000 }
gfCNCPoint5[26832] = {X 330.2784, Y 83.5896, Z -8.0000, A 0.000, B 0.000, C 0.000 }
gfCNCPoint5[26833] = {X 330.5997, Y 83.6700, Z -8.0000, A 0.000, B 0.000, C 0.000 }
gfCNCPoint5[26834] = {X 330.9235, Y 83.7402, Z -8.0000, A 0.000, B 0.000, C 0.000 }
gfCNCPoint5[26835] = {X 333.6940, Y 84.2386, Z -8.0000, A 0.000, B 0.000, C 0.000 }
gfCNCPoint5[26836] = {X 336.4899, Y 84.5666, Z -8.0000, A 0.000, B 0.000, C 0.000 }
gfCNCPoint5[26837] = {X 340.6971, Y 84.8495, Z -8.0000, A 0.000, B 0.000, C 0.000 }
gfCNCPoint5[26838] = {X 344.9112, Y 84.9969, Z -8.0000, A 0.000, B 0.000, C 0.000 }
gfCNCPoint5[26839] = {X 349.1279, Y 85.0087, Z -8.0000, A 0.000, B 0.000, C 0.000 }
gfCNCPoint5[26840] = {X 353.0976, Y 84.9447, Z -8.0000, A 0.000, B 0.000, C 0.000 }
gfCNCPoint5[26841] = {X 357.0623, Y 84.7362, Z -8.0000, A 0.000, B 0.000, C 0.000 }
gfCNCPoint5[26842] = {X 361.0167, Y 84.3835, Z -8.0000, A 0.000, B 0.000, C 0.000 }
gfCNCPoint5[26843] = {X 363.3024, Y 84.0496, Z -8.0000, A 0.000, B 0.000, C 0.000 }
gfCNCPoint5[26844] = {X 365.5587, Y 83.5544, Z -8.0000, A 0.000, B 0.000, C 0.000 }
gfCNCPoint5[26845] = {X 365.5578, Y 66.5605, Z -8.0000, A 0.000, B 0.000, C 0.000 }
gfCNCPoint5[26846] = {X 364.4837, Y 65.5826, Z -8.0000, A 0.000, B 0.000, C 0.000 }
gfCNCPoint5[26847] = {X 363.5680, Y 64.4549, Z -8.0000, A 0.000, B 0.000, C 0.000 }
gfCNCPoint5[26848] = {X 362.8314, Y 63.2029, Z -8.0000, A 0.000, B 0.000, C 0.000 }
gfCNCPoint5[26849] = {X 362.2904, Y 61.8548, Z -8.0000, A 0.000, B 0.000, C 0.000 }
gfCNCPoint5[26850] = {X 361.9573, Y 60.4408, Z -8.0000, A 0.000, B 0.000, C 0.000 }
gfCNCPoint5[26851] = {X 361.8395, Y 58.9930, Z -8.0000, A 0.000, B 0.000, C 0.000 }
gfCNCPoint5[26852] = {X 361.8393, Y 58.0000, Z -8.0000, A 0.000, B 0.000, C 0.000 }
gfCNCPoint5[26853] = {X 361.9152, Y 56.7904, Z -8.0000, A 0.000, B 0.000, C 0.000 }
gfCNCPoint5[26854] = {X 362.1416, Y 55.5998, Z -8.0000, A 0.000, B 0.000, C 0.000 }
gfCNCPoint5[26855] = {X 362.5726, Y 54.3043, Z -8.0000, A 0.000, B 0.000, C 0.000 }
gfCNCPoint5[26856] = {X 363.1816, Y 53.0822, Z -8.0000, A 0.000, B 0.000, C 0.000 }
gfCNCPoint5[26857] = {X 363.9564, Y 51.9580, Z -8.0000, A 0.000, B 0.000, C 0.000 }
gfCNCPoint5[26858] = {X 364.8818, Y 50.9540, Z -8.0000, A 0.000, B 0.000, C 0.000 }
gfCNCPoint5[26859] = {X 365.9392, Y 50.0902, Z -8.0000, A 0.000, B 0.000, C 0.000 }
gfCNCPoint5[26860] = {X 367.1076, Y 49.3838, Z -8.0000, A 0.000, B 0.000, C 0.000 }
gfCNCPoint5[26861] = {X 368.3638, Y 48.8487, Z -8.0000, A 0.000, B 0.000, C 0.000 }
gfCNCPoint5[26862] = {X 369.6828, Y 48.4958, Z -8.0000, A 0.000, B 0.000, C 0.000 }
gfCNCPoint5[26863] = {X 371.0383, Y 48.3320, Z -8.0000, A 0.000, B 0.000, C 0.000 }
gfCNCPoint5[26864] = {X 371.2787, Y 48.3230, Z -8.0000, A 0.000, B 0.000, C 0.000 }
gfCNCPoint5[26865] = {X 371.5193, Y 48.3200, Z -8.0000, A 0.000, B 0.000, C 0.000 }
gfCNCPoint5[26866] = {X 388.0597, Y 48.3200, Z -8.0000, A 0.000, B 0.000, C 0.000 }
gfCNCPoint5[26867] = {X 389.4419, Y 48.4192, Z -8.0000, A 0.000, B 0.000, C 0.000 }
gfCNCPoint5[26868] = {X 390.7958, Y 48.7147, Z -8.0000, A 0.000, B 0.000, C 0.000 }
gfCNCPoint5[26869] = {X 392.0936, Y 49.2006, Z -8.0000, A 0.000, B 0.000, C 0.000 }
gfCNCPoint5[26870] = {X 393.3087, Y 49.8667, Z -8.0000, A 0.000, B 0.000, C 0.000 }
gfCNCPoint5[26871] = {X 394.5333, Y 49.1962, Z -8.0000, A 0.000, B 0.000, C 0.000 }
gfCNCPoint5[26872] = {X 395.8416, Y 48.7089, Z -8.0000, A 0.000, B 0.000, C 0.000 }
gfCNCPoint5[26873] = {X 397.1858, Y 48.4177, Z -8.0000, A 0.000, B 0.000, C 0.000 }
gfCNCPoint5[26874] = {X 398.5577, Y 48.3200, Z -8.0000, A 0.000, B 0.000, C 0.000 }
gfCNCPoint5[26875] = {X 398.7346, Y 48.3200, Z -8.0000, A 0.000, B 0.000, C 0.000 }
gfCNCPoint5[26876] = {X 398.1859, Y 47.6069, Z -8.0000, A 0.000, B 0.000, C 0.000 }
gfCNCPoint5[26877] = {X 397.7774, Y 46.8051, Z -8.0000, A 0.000, B 0.000, C 0.000 }
gfCNCPoint5[26878] = {X 397.5230, Y 45.9420, Z -8.0000, A 0.000, B 0.000, C 0.000 }
gfCNCPoint5[26879] = {X 397.4561, Y 45.4921, Z -8.0000, A 0.000, B 0.000, C 0.000 }
gfCNCPoint5[26880] = {X 397.4314, Y 45.0378, Z -8.0000, A 0.000, B 0.000, C 0.000 }
gfCNCPoint5[26881] = {X 397.4316, Y 44.1455, Z -8.0000, A 0.000, B 0.000, C 0.000 }
gfCNCPoint5[26882] = {X 397.5413, Y 43.1779, Z -8.0000, A 0.000, B 0.000, C 0.000 }
gfCNCPoint5[26883] = {X 397.8410, Y 42.2514, Z -8.0000, A 0.000, B 0.000, C 0.000 }
gfCNCPoint5[26884] = {X 398.3186, Y 41.4028, Z -8.0000, A 0.000, B 0.000, C 0.000 }
gfCNCPoint5[26885] = {X 398.9552, Y 40.6660, Z -8.0000, A 0.000, B 0.000, C 0.000 }
gfCNCPoint5[26886] = {X 398.9552, Y 31.8260, Z -8.0000, A 0.000, B 0.000, C 0.000 }
gfCNCPoint5[26887] = {X 392.9491, Y 21.3815, Z -8.0000, A 0.000, B 0.000, C 0.000 }
gfCNCPoint5[26888] = {X 392.1065, Y 19.9495, Z -8.0000, A 0.000, B 0.000, C 0.000 }
gfCNCPoint5[26889] = {X 391.2354, Y 18.5346, Z -8.0000, A 0.000, B 0.000, C 0.000 }
gfCNCPoint5[26890] = {X 390.8255, Y 17.9610, Z -8.0000, A 0.000, B 0.000, C 0.000 }
gfCNCPoint5[26891] = {X 390.3515, Y 17.4391, Z -8.0000, A 0.000, B 0.000, C 0.000 }
gfCNCPoint5[26892] = {X 389.5418, Y 16.9833, Z -8.0000, A 0.000, B 0.000, C 0.000 }
gfCNCPoint5[26893] = {X 388.8332, Y 16.3823, Z -8.0000, A 0.000, B 0.000, C 0.000 }
gfCNCPoint5[26894] = {X 388.2513, Y 15.6579, Z -8.0000, A 0.000, B 0.000, C 0.000 }
gfCNCPoint5[26895] = {X 387.8173, Y 14.8363, Z -8.0000, A 0.000, B 0.000, C 0.000 }
gfCNCPoint5[26896] = {X 387.5469, Y 13.9473, Z -8.0000, A 0.000, B 0.000, C 0.000 }
gfCNCPoint5[26897] = {X 387.4498, Y 13.0232, Z -8.0000, A 0.000, B 0.000, C 0.000 }
gfCNCPoint5[26898] = {X 387.4496, Y 12.1868, Z -8.0000, A 0.000, B 0.000, C 0.000 }
gfCNCPoint5[26899] = {X 387.5362, Y 11.2717, Z -8.0000, A 0.000, B 0.000, C 0.000 }
gfCNCPoint5[26900] = {X 387.7929, Y 10.3890, Z -8.0000, A 0.000, B 0.000, C 0.000 }
gfCNCPoint5[26901] = {X 388.2376, Y 9.5279, Z -8.0000, A 0.000, B 0.000, C 0.000 }
gfCNCPoint5[26902] = {X 388.8437, Y 8.7718, Z -8.0000, A 0.000, B 0.000, C 0.000 }
gfCNCPoint5[26903] = {X 389.5873, Y 8.1502, Z -8.0000, A 0.000, B 0.000, C 0.000 }
gfCNCPoint5[26904] = {X 390.4390, Y 7.6879, Z -8.0000, A 0.000, B 0.000, C 0.000 }
gfCNCPoint5[26905] = {X 391.3653, Y 7.4030, Z -8.0000, A 0.000, B 0.000, C 0.000 }
gfCNCPoint5[26906] = {X 392.3296, Y 7.3068, Z -8.0000, A 0.000, B 0.000, C 0.000 }
gfCNCPoint5[26907] = {X 399.1118, Y 7.3068, Z -8.0000, A 0.000, B 0.000, C 0.000 }
gfCNCPoint5[26908] = {X 400.0638, Y 7.4006, Z -8.0000, A 0.000, B 0.000, C 0.000 }
gfCNCPoint5[26909] = {X 400.9793, Y 7.6783, Z -8.0000, A 0.000, B 0.000, C 0.000 }
gfCNCPoint5[26910] = {X 401.8229, Y 8.1292, Z -8.0000, A 0.000, B 0.000, C 0.000 }
gfCNCPoint5[26911] = {X 402.5624, Y 8.7361, Z -8.0000, A 0.000, B 0.000, C 0.000 }
gfCNCPoint5[26912] = {X 403.1693, Y 9.4756, Z -8.0000, A 0.000, B 0.000, C 0.000 }
gfCNCPoint5[26913] = {X 403.6203, Y 10.3193, Z -8.0000, A 0.000, B 0.000, C 0.000 }
gfCNCPoint5[26914] = {X 403.8980, Y 11.2348, Z -8.0000, A 0.000, B 0.000, C 0.000 }
gfCNCPoint5[26915] = {X 403.9918, Y 12.1868, Z -8.0000, A 0.000, B 0.000, C 0.000 }
gfCNCPoint5[26916] = {X 403.9915, Y 13.0237, Z -8.0000, A 0.000, B 0.000, C 0.000 }
gfCNCPoint5[26917] = {X 403.9016, Y 13.9115, Z -8.0000, A 0.000, B 0.000, C 0.000 }
gfCNCPoint5[26918] = {X 403.6516, Y 14.7680, Z -8.0000, A 0.000, B 0.000, C 0.000 }
gfCNCPoint5[26919] = {X 405.3641, Y 17.7415, Z -8.0000, A 0.000, B 0.000, C 0.000 }
gfCNCPoint5[26920] = {X 407.2441, Y 14.6964, Z -8.0000, A 0.000, B 0.000, C 0.000 }
gfCNCPoint5[26921] = {X 407.0141, Y 13.8719, Z -8.0000, A 0.000, B 0.000, C 0.000 }
gfCNCPoint5[26922] = {X 406.9317, Y 13.0199, Z -8.0000, A 0.000, B 0.000, C 0.000 }
gfCNCPoint5[26923] = {X 406.9315, Y 12.1868, Z -8.0000, A 0.000, B 0.000, C 0.000 }
gfCNCPoint5[26924] = {X 407.0253, Y 11.2348, Z -8.0000, A 0.000, B 0.000, C 0.000 }
gfCNCPoint5[26925] = {X 407.3030, Y 10.3193, Z -8.0000, A 0.000, B 0.000, C 0.000 }
gfCNCPoint5[26926] = {X 407.7540, Y 9.4756, Z -8.0000, A 0.000, B 0.000, C 0.000 }
gfCNCPoint5[26927] = {X 408.3609, Y 8.7361, Z -8.0000, A 0.000, B 0.000, C 0.000 }
gfCNCPoint5[26928] = {X 409.1004, Y 8.1292, Z -8.0000, A 0.000, B 0.000, C 0.000 }
gfCNCPoint5[26929] = {X 409.9440, Y 7.6783, Z -8.0000, A 0.000, B 0.000, C 0.000 }
gfCNCPoint5[26930] = {X 410.8595, Y 7.4006, Z -8.0000, A 0.000, B 0.000, C 0.000 }
gfCNCPoint5[26931] = {X 411.8115, Y 7.3068, Z -8.0000, A 0.000, B 0.000, C 0.000 }
gfCNCPoint5[26932] = {X 419.3245, Y 7.3068, Z -8.0000, A 0.000, B 0.000, C 0.000 }
gfCNCPoint5[26933] = {X 420.2888, Y 7.4030, Z -8.0000, A 0.000, B 0.000, C 0.000 }
gfCNCPoint5[26934] = {X 421.2151, Y 7.6879, Z -8.0000, A 0.000, B 0.000, C 0.000 }
gfCNCPoint5[26935] = {X 422.0668, Y 8.1502, Z -8.0000, A 0.000, B 0.000, C 0.000 }
gfCNCPoint5[26936] = {X 422.8104, Y 8.7718, Z -8.0000, A 0.000, B 0.000, C 0.000 }
gfCNCPoint5[26937] = {X 423.4165, Y 9.5279, Z -8.0000, A 0.000, B 0.000, C 0.000 }
gfCNCPoint5[26938] = {X 423.8612, Y 10.3890, Z -8.0000, A 0.000, B 0.000, C 0.000 }
gfCNCPoint5[26939] = {X 424.1179, Y 11.2717, Z -8.0000, A 0.000, B 0.000, C 0.000 }
gfCNCPoint5[26940] = {X 424.2045, Y 12.1868, Z -8.0000, A 0.000, B 0.000, C 0.000 }
gfCNCPoint5[26941] = {X 424.2045, Y 12.9780, Z -8.0000, A 0.000, B 0.000, C 0.000 }
gfCNCPoint5[26942] = {X 424.1066, Y 13.9309, Z -8.0000, A 0.000, B 0.000, C 0.000 }
gfCNCPoint5[26943] = {X 423.8266, Y 14.8469, Z -8.0000, A 0.000, B 0.000, C 0.000 }
gfCNCPoint5[26944] = {X 423.3751, Y 15.6917, Z -8.0000, A 0.000, B 0.000, C 0.000 }
gfCNCPoint5[26945] = {X 422.7690, Y 16.4334, Z -8.0000, A 0.000, B 0.000, C 0.000 }
gfCNCPoint5[26946] = {X 422.0312, Y 17.0443, Z -8.0000, A 0.000, B 0.000, C 0.000 }
gfCNCPoint5[26947] = {X 421.1893, Y 17.5012, Z -8.0000, A 0.000, B 0.000, C 0.000 }
gfCNCPoint5[26948] = {X 420.5414, Y 18.3845, Z -8.0000, A 0.000, B 0.000, C 0.000 }
gfCNCPoint5[26949] = {X 419.9525, Y 19.3082, Z -8.0000, A 0.000, B 0.000, C 0.000 }
gfCNCPoint5[26950] = {X 414.1632, Y 28.6202, Z -8.0000, A 0.000, B 0.000, C 0.000 }
gfCNCPoint5[26951] = {X 422.3160, Y 33.6889, Z -8.0000, A 0.000, B 0.000, C 0.000 }
gfCNCPoint5[26952] = {X 421.8968, Y 34.3631, Z -8.0000, A 0.000, B 0.000, C 0.000 }
gfCNCPoint5[26953] = {X 422.1490, Y 34.0980, Z -8.0000, A 0.000, B 0.000, C 0.000 }
gfCNCPoint5[26954] = {X 422.4077, Y 33.8394, Z -8.0000, A 0.000, B 0.000, C 0.000 }
gfCNCPoint5[26955] = {X 422.3617, Y 33.7642, Z -8.0000, A 0.000, B 0.000, C 0.000 }
gfCNCPoint5[26956] = {X 422.3160, Y 33.6889, Z -8.0000, A 0.000, B 0.000, C 0.000 }
gfCNCPoint5[26957] = {X 420.2778, Y 32.4217, Z -8.0000, A 0.000, B 0.000, C 0.000 }
gfCNCPoint5[26958] = {X 419.3084, Y 33.9810, Z -8.0000, A 0.000, B 0.000, C 0.000 }
gfCNCPoint5[26959] = {X 419.3087, Y 38.3383, Z -8.0000, A 0.000, B 0.000, C 0.000 }
gfCNCPoint5[26960] = {X 419.9590, Y 39.7074, Z -8.0000, A 0.000, B 0.000, C 0.000 }
gfCNCPoint5[26961] = {X 420.4344, Y 41.1465, Z -8.0000, A 0.000, B 0.000, C 0.000 }
gfCNCPoint5[26962] = {X 420.6284, Y 41.1585, Z -8.0000, A 0.000, B 0.000, C 0.000 }
gfCNCPoint5[26963] = {X 420.8222, Y 41.1728, Z -8.0000, A 0.000, B 0.000, C 0.000 }
gfCNCPoint5[26964] = {X 421.2848, Y 39.7566, Z -8.0000, A 0.000, B 0.000, C 0.000 }
gfCNCPoint5[26965] = {X 421.9183, Y 38.4081, Z -8.0000, A 0.000, B 0.000, C 0.000 }
gfCNCPoint5[26966] = {X 422.7129, Y 37.1478, Z -8.0000, A 0.000, B 0.000, C 0.000 }
gfCNCPoint5[26967] = {X 423.6567, Y 35.9950, Z -8.0000, A 0.000, B 0.000, C 0.000 }
gfCNCPoint5[26968] = {X 424.3435, Y 35.3115, Z -8.0000, A 0.000, B 0.000, C 0.000 }
gfCNCPoint5[26969] = {X 425.0829, Y 34.6852, Z -8.0000, A 0.000, B 0.000, C 0.000 }
gfCNCPoint5[26970] = {X 425.4255, Y 34.0144, Z -8.0000, A 0.000, B 0.000, C 0.000 }
gfCNCPoint5[26971] = {X 424.8786, Y 33.2443, Z -8.0000, A 0.000, B 0.000, C 0.000 }
gfCNCPoint5[26972] = {X 424.3704, Y 32.4481, Z -8.0000, A 0.000, B 0.000, C 0.000 }
gfCNCPoint5[26973] = {X 423.3893, Y 30.6026, Z -8.0000, A 0.000, B 0.000, C 0.000 }
gfCNCPoint5[26974] = {X 422.6159, Y 28.6609, Z -8.0000, A 0.000, B 0.000, C 0.000 }
gfCNCPoint5[26975] = {X 420.2778, Y 32.4217, Z -8.0000, A 0.000, B 0.000, C 0.000 }
gfCNCPoint5[26976] = {X 418.2396, Y 31.1546, Z -8.0000, A 0.000, B 0.000, C 0.000 }
gfCNCPoint5[26977] = {X 416.9083, Y 33.2959, Z -8.0000, A 0.000, B 0.000, C 0.000 }
gfCNCPoint5[26978] = {X 416.9087, Y 38.9949, Z -8.0000, A 0.000, B 0.000, C 0.000 }
gfCNCPoint5[26979] = {X 417.4900, Y 40.0482, Z -8.0000, A 0.000, B 0.000, C 0.000 }
gfCNCPoint5[26980] = {X 417.9377, Y 41.1649, Z -8.0000, A 0.000, B 0.000, C 0.000 }
gfCNCPoint5[26981] = {X 418.2452, Y 42.3280, Z -8.0000, A 0.000, B 0.000, C 0.000 }
gfCNCPoint5[26982] = {X 418.4079, Y 43.5200, Z -8.0000, A 0.000, B 0.000, C 0.000 }
gfCNCPoint5[26983] = {X 419.4886, Y 43.5200, Z -8.0000, A 0.000, B 0.000, C 0.000 }
gfCNCPoint5[26984] = {X 421.1752, Y 43.6186, Z -8.0000, A 0.000, B 0.000, C 0.000 }
gfCNCPoint5[26985] = {X 422.8389, Y 43.9129, Z -8.0000, A 0.000, B 0.000, C 0.000 }
gfCNCPoint5[26986] = {X 423.0005, Y 42.4234, Z -8.0000, A 0.000, B 0.000, C 0.000 }
gfCNCPoint5[26987] = {X 423.3900, Y 40.9766, Z -8.0000, A 0.000, B 0.000, C 0.000 }
gfCNCPoint5[26988] = {X 423.9980, Y 39.6073, Z -8.0000, A 0.000, B 0.000, C 0.000 }
gfCNCPoint5[26989] = {X 424.8102, Y 38.3482, Z -8.0000, A 0.000, B 0.000, C 0.000 }
gfCNCPoint5[26990] = {X 425.8068, Y 37.2295, Z -8.0000, A 0.000, B 0.000, C 0.000 }
gfCNCPoint5[26991] = {X 426.9642, Y 36.2780, Z -8.0000, A 0.000, B 0.000, C 0.000 }
gfCNCPoint5[26992] = {X 428.2759, Y 33.7106, Z -8.0000, A 0.000, B 0.000, C 0.000 }
gfCNCPoint5[26993] = {X 427.2122, Y 32.3936, Z -8.0000, A 0.000, B 0.000, C 0.000 }
gfCNCPoint5[26994] = {X 426.2874, Y 30.9757, Z -8.0000, A 0.000, B 0.000, C 0.000 }
gfCNCPoint5[26995] = {X 425.5109, Y 29.4714, Z -8.0000, A 0.000, B 0.000, C 0.000 }
gfCNCPoint5[26996] = {X 424.8908, Y 27.8961, Z -8.0000, A 0.000, B 0.000, C 0.000 }
gfCNCPoint5[26997] = {X 424.8189, Y 27.6772, Z -8.0000, A 0.000, B 0.000, C 0.000 }
gfCNCPoint5[26998] = {X 424.7500, Y 27.4573, Z -8.0000, A 0.000, B 0.000, C 0.000 }
gfCNCPoint5[26999] = {X 424.3069, Y 25.7014, Z -8.0000, A 0.000, B 0.000, C 0.000 }
gfCNCPoint5[27000] = {X 424.0105, Y 23.9149, Z -8.0000, A 0.000, B 0.000, C 0.000 }
gfCNCPoint5[27001] = {X 423.8627, Y 22.1100, Z -8.0000, A 0.000, B 0.000, C 0.000 }
gfCNCPoint5[27002] = {X 418.2396, Y 31.1546, Z -8.0000, A 0.000, B 0.000, C 0.000 }
gfCNCPoint5[27003] = {X 416.2014, Y 29.8874, Z -8.0000, A 0.000, B 0.000, C 0.000 }
gfCNCPoint5[27004] = {X 414.5083, Y 32.6107, Z -8.0000, A 0.000, B 0.000, C 0.000 }
gfCNCPoint5[27005] = {X 414.5087, Y 39.7462, Z -8.0000, A 0.000, B 0.000, C 0.000 }
gfCNCPoint5[27006] = {X 415.1574, Y 40.7516, Z -8.0000, A 0.000, B 0.000, C 0.000 }
gfCNCPoint5[27007] = {X 415.6355, Y 41.8484, Z -8.0000, A 0.000, B 0.000, C 0.000 }
gfCNCPoint5[27008] = {X 415.9305, Y 43.0080, Z -8.0000, A 0.000, B 0.000, C 0.000 }
gfCNCPoint5[27009] = {X 416.0347, Y 44.1999, Z -8.0000, A 0.000, B 0.000, C 0.000 }
gfCNCPoint5[27010] = {X 416.0347, Y 45.0000, Z -8.0000, A 0.000, B 0.000, C 0.000 }
gfCNCPoint5[27011] = {X 416.0201, Y 45.4609, Z -8.0000, A 0.000, B 0.000, C 0.000 }
gfCNCPoint5[27012] = {X 415.9763, Y 45.9200, Z -8.0000, A 0.000, B 0.000, C 0.000 }
gfCNCPoint5[27013] = {X 419.4886, Y 45.9200, Z -8.0000, A 0.000, B 0.000, C 0.000 }
gfCNCPoint5[27014] = {X 420.8957, Y 46.0022, Z -8.0000, A 0.000, B 0.000, C 0.000 }
gfCNCPoint5[27015] = {X 422.2836, Y 46.2478, Z -8.0000, A 0.000, B 0.000, C 0.000 }
gfCNCPoint5[27016] = {X 423.4822, Y 46.5992, Z -8.0000, A 0.000, B 0.000, C 0.000 }
gfCNCPoint5[27017] = {X 424.6380, Y 47.0725, Z -8.0000, A 0.000, B 0.000, C 0.000 }
gfCNCPoint5[27018] = {X 425.7388, Y 47.6626, Z -8.0000, A 0.000, B 0.000, C 0.000 }
gfCNCPoint5[27019] = {X 425.4600, Y 46.7984, Z -8.0000, A 0.000, B 0.000, C 0.000 }
gfCNCPoint5[27020] = {X 425.2910, Y 45.9063, Z -8.0000, A 0.000, B 0.000, C 0.000 }
gfCNCPoint5[27021] = {X 425.2344, Y 45.0000, Z -8.0000, A 0.000, B 0.000, C 0.000 }
gfCNCPoint5[27022] = {X 425.2344, Y 44.2089, Z -8.0000, A 0.000, B 0.000, C 0.000 }
gfCNCPoint5[27023] = {X 425.2353, Y 44.0976, Z -8.0000, A 0.000, B 0.000, C 0.000 }
gfCNCPoint5[27024] = {X 425.2378, Y 43.9863, Z -8.0000, A 0.000, B 0.000, C 0.000 }
gfCNCPoint5[27025] = {X 425.3770, Y 42.7748, Z -8.0000, A 0.000, B 0.000, C 0.000 }
gfCNCPoint5[27026] = {X 425.7165, Y 41.6036, Z -8.0000, A 0.000, B 0.000, C 0.000 }
gfCNCPoint5[27027] = {X 426.2468, Y 40.5054, Z -8.0000, A 0.000, B 0.000, C 0.000 }
gfCNCPoint5[27028] = {X 426.9528, Y 39.5112, Z -8.0000, A 0.000, B 0.000, C 0.000 }
gfCNCPoint5[27029] = {X 427.8150, Y 38.6488, Z -8.0000, A 0.000, B 0.000, C 0.000 }
gfCNCPoint5[27030] = {X 428.8090, Y 37.9424, Z -8.0000, A 0.000, B 0.000, C 0.000 }
gfCNCPoint5[27031] = {X 431.2065, Y 33.2495, Z -8.0000, A 0.000, B 0.000, C 0.000 }
gfCNCPoint5[27032] = {X 430.1005, Y 32.1504, Z -8.0000, A 0.000, B 0.000, C 0.000 }
gfCNCPoint5[27033] = {X 429.1209, Y 30.9374, Z -8.0000, A 0.000, B 0.000, C 0.000 }
gfCNCPoint5[27034] = {X 428.2792, Y 29.6248, Z -8.0000, A 0.000, B 0.000, C 0.000 }
gfCNCPoint5[27035] = {X 427.5854, Y 28.2284, Z -8.0000, A 0.000, B 0.000, C 0.000 }
gfCNCPoint5[27036] = {X 427.0480, Y 26.7648, Z -8.0000, A 0.000, B 0.000, C 0.000 }
gfCNCPoint5[27037] = {X 426.6549, Y 25.2044, Z -8.0000, A 0.000, B 0.000, C 0.000 }
gfCNCPoint5[27038] = {X 426.3919, Y 23.6169, Z -8.0000, A 0.000, B 0.000, C 0.000 }
gfCNCPoint5[27039] = {X 426.2607, Y 22.0132, Z -8.0000, A 0.000, B 0.000, C 0.000 }
gfCNCPoint5[27040] = {X 426.2908, Y 19.8890, Z -8.0000, A 0.000, B 0.000, C 0.000 }
gfCNCPoint5[27041] = {X 426.5520, Y 17.7807, Z -8.0000, A 0.000, B 0.000, C 0.000 }
gfCNCPoint5[27042] = {X 427.0409, Y 15.7133, Z -8.0000, A 0.000, B 0.000, C 0.000 }
gfCNCPoint5[27043] = {X 427.6625, Y 14.0032, Z -8.0000, A 0.000, B 0.000, C 0.000 }
gfCNCPoint5[27044] = {X 428.4894, Y 12.3823, Z -8.0000, A 0.000, B 0.000, C 0.000 }
gfCNCPoint5[27045] = {X 429.5090, Y 10.8753, Z -8.0000, A 0.000, B 0.000, C 0.000 }
gfCNCPoint5[27046] = {X 430.7059, Y 9.5048, Z -8.0000, A 0.000, B 0.000, C 0.000 }
gfCNCPoint5[27047] = {X 426.0924, Y 9.5048, Z -8.0000, A 0.000, B 0.000, C 0.000 }
gfCNCPoint5[27048] = {X 426.3754, Y 10.3749, Z -8.0000, A 0.000, B 0.000, C 0.000 }
gfCNCPoint5[27049] = {X 426.5470, Y 11.2737, Z -8.0000, A 0.000, B 0.000, C 0.000 }
gfCNCPoint5[27050] = {X 426.6045, Y 12.1868, Z -8.0000, A 0.000, B 0.000, C 0.000 }
gfCNCPoint5[27051] = {X 426.6044, Y 12.9907, Z -8.0000, A 0.000, B 0.000, C 0.000 }
gfCNCPoint5[27052] = {X 426.4812, Y 14.2917, Z -8.0000, A 0.000, B 0.000, C 0.000 }
gfCNCPoint5[27053] = {X 426.1292, Y 15.5503, Z -8.0000, A 0.000, B 0.000, C 0.000 }
gfCNCPoint5[27054] = {X 425.5595, Y 16.7265, Z -8.0000, A 0.000, B 0.000, C 0.000 }
gfCNCPoint5[27055] = {X 424.7903, Y 17.7831, Z -8.0000, A 0.000, B 0.000, C 0.000 }
gfCNCPoint5[27056] = {X 423.8459, Y 18.6864, Z -8.0000, A 0.000, B 0.000, C 0.000 }
gfCNCPoint5[27057] = {X 422.7562, Y 19.4079, Z -8.0000, A 0.000, B 0.000, C 0.000 }
gfCNCPoint5[27058] = {X 422.3665, Y 19.9718, Z -8.0000, A 0.000, B 0.000, C 0.000 }
gfCNCPoint5[27059] = {X 422.0042, Y 20.5537, Z -8.0000, A 0.000, B 0.000, C 0.000 }
gfCNCPoint5[27060] = {X 416.2014, Y 29.8874, Z -8.0000, A 0.000, B 0.000, C 0.000 }
gfCNCPoint5[27061] = {X 414.1632, Y 28.6202, Z -8.0000, A 0.000, B 0.000, C 0.000 }
gfCNCPoint5[27062] = {X 412.1082, Y 31.9255, Z -8.0000, A 0.000, B 0.000, C 0.000 }
gfCNCPoint5[27063] = {X 412.1088, Y 40.6512, Z -8.0000, A 0.000, B 0.000, C 0.000 }
gfCNCPoint5[27064] = {X 412.7506, Y 41.4078, Z -8.0000, A 0.000, B 0.000, C 0.000 }
gfCNCPoint5[27065] = {X 413.2302, Y 42.2763, Z -8.0000, A 0.000, B 0.000, C 0.000 }
gfCNCPoint5[27066] = {X 413.5289, Y 43.2224, Z -8.0000, A 0.000, B 0.000, C 0.000 }
gfCNCPoint5[27067] = {X 413.6347, Y 44.2088, Z -8.0000, A 0.000, B 0.000, C 0.000 }
gfCNCPoint5[27068] = {X 413.6347, Y 45.0000, Z -8.0000, A 0.000, B 0.000, C 0.000 }
gfCNCPoint5[27069] = {X 413.6249, Y 45.3090, Z -8.0000, A 0.000, B 0.000, C 0.000 }
gfCNCPoint5[27070] = {X 413.5956, Y 45.6167, Z -8.0000, A 0.000, B 0.000, C 0.000 }
gfCNCPoint5[27071] = {X 413.3652, Y 46.5992, Z -8.0000, A 0.000, B 0.000, C 0.000 }
gfCNCPoint5[27072] = {X 412.9377, Y 47.5134, Z -8.0000, A 0.000, B 0.000, C 0.000 }
gfCNCPoint5[27073] = {X 412.3313, Y 48.3200, Z -8.0000, A 0.000, B 0.000, C 0.000 }
gfCNCPoint5[27074] = {X 411.9795, Y 47.9934, Z -8.0000, A 0.000, B 0.000, C 0.000 }
gfCNCPoint5[27075] = {X 411.3003, Y 48.5889, Z -8.0000, A 0.000, B 0.000, C 0.000 }
gfCNCPoint5[27076] = {X 410.5138, Y 49.0331, Z -8.0000, A 0.000, B 0.000, C 0.000 }
gfCNCPoint5[27077] = {X 409.6532, Y 49.3073, Z -8.0000, A 0.000, B 0.000, C 0.000 }
gfCNCPoint5[27078] = {X 408.7547, Y 49.4000, Z -8.0000, A 0.000, B 0.000, C 0.000 }
gfCNCPoint5[27079] = {X 402.3112, Y 49.4000, Z -8.0000, A 0.000, B 0.000, C 0.000 }
gfCNCPoint5[27080] = {X 401.3321, Y 49.2897, Z -8.0000, A 0.000, B 0.000, C 0.000 }
gfCNCPoint5[27081] = {X 400.4021, Y 48.9643, Z -8.0000, A 0.000, B 0.000, C 0.000 }
gfCNCPoint5[27082] = {X 399.5678, Y 48.4401, Z -8.0000, A 0.000, B 0.000, C 0.000 }
gfCNCPoint5[27083] = {X 398.8711, Y 47.7433, Z -8.0000, A 0.000, B 0.000, C 0.000 }
gfCNCPoint5[27084] = {X 398.3469, Y 46.9091, Z -8.0000, A 0.000, B 0.000, C 0.000 }
gfCNCPoint5[27085] = {X 398.0215, Y 45.9791, Z -8.0000, A 0.000, B 0.000, C 0.000 }
gfCNCPoint5[27086] = {X 397.9112, Y 45.0000, Z -8.0000, A 0.000, B 0.000, C 0.000 }
gfCNCPoint5[27087] = {X 397.9116, Y 44.1518, Z -8.0000, A 0.000, B 0.000, C 0.000 }
gfCNCPoint5[27088] = {X 398.0215, Y 43.2300, Z -8.0000, A 0.000, B 0.000, C 0.000 }
gfCNCPoint5[27089] = {X 398.3223, Y 42.3519, Z -8.0000, A 0.000, B 0.000, C 0.000 }
gfCNCPoint5[27090] = {X 398.8006, Y 41.5563, Z -8.0000, A 0.000, B 0.000, C 0.000 }
gfCNCPoint5[27091] = {X 399.4352, Y 40.8789, Z -8.0000, A 0.000, B 0.000, C 0.000 }
gfCNCPoint5[27092] = {X 399.4352, Y 31.6979, Z -8.0000, A 0.000, B 0.000, C 0.000 }
gfCNCPoint5[27093] = {X 393.3653, Y 21.1422, Z -8.0000, A 0.000, B 0.000, C 0.000 }
gfCNCPoint5[27094] = {X 392.5177, Y 19.7019, Z -8.0000, A 0.000, B 0.000, C 0.000 }
gfCNCPoint5[27095] = {X 391.6416, Y 18.2789, Z -8.0000, A 0.000, B 0.000, C 0.000 }
gfCNCPoint5[27096] = {X 391.1705, Y 17.6244, Z -8.0000, A 0.000, B 0.000, C 0.000 }
gfCNCPoint5[27097] = {X 390.6221, Y 17.0332, Z -8.0000, A 0.000, B 0.000, C 0.000 }
gfCNCPoint5[27098] = {X 389.8674, Y 16.6246, Z -8.0000, A 0.000, B 0.000, C 0.000 }
gfCNCPoint5[27099] = {X 389.2063, Y 16.0772, Z -8.0000, A 0.000, B 0.000, C 0.000 }
gfCNCPoint5[27100] = {X 388.6640, Y 15.4118, Z -8.0000, A 0.000, B 0.000, C 0.000 }
gfCNCPoint5[27101] = {X 388.2613, Y 14.6539, Z -8.0000, A 0.000, B 0.000, C 0.000 }
gfCNCPoint5[27102] = {X 388.0133, Y 13.8322, Z -8.0000, A 0.000, B 0.000, C 0.000 }
gfCNCPoint5[27103] = {X 387.9296, Y 12.9780, Z -8.0000, A 0.000, B 0.000, C 0.000 }
gfCNCPoint5[27104] = {X 387.9296, Y 12.1868, Z -8.0000, A 0.000, B 0.000, C 0.000 }
gfCNCPoint5[27105] = {X 388.0399, Y 11.2077, Z -8.0000, A 0.000, B 0.000, C 0.000 }
gfCNCPoint5[27106] = {X 388.3654, Y 10.2777, Z -8.0000, A 0.000, B 0.000, C 0.000 }
gfCNCPoint5[27107] = {X 388.8896, Y 9.4435, Z -8.0000, A 0.000, B 0.000, C 0.000 }
gfCNCPoint5[27108] = {X 389.5863, Y 8.7468, Z -8.0000, A 0.000, B 0.000, C 0.000 }
gfCNCPoint5[27109] = {X 390.4205, Y 8.2226, Z -8.0000, A 0.000, B 0.000, C 0.000 }
gfCNCPoint5[27110] = {X 391.3505, Y 7.8971, Z -8.0000, A 0.000, B 0.000, C 0.000 }
gfCNCPoint5[27111] = {X 392.3296, Y 7.7868, Z -8.0000, A 0.000, B 0.000, C 0.000 }
gfCNCPoint5[27112] = {X 399.1118, Y 7.7868, Z -8.0000, A 0.000, B 0.000, C 0.000 }
gfCNCPoint5[27113] = {X 400.0909, Y 7.8971, Z -8.0000, A 0.000, B 0.000, C 0.000 }
gfCNCPoint5[27114] = {X 401.0208, Y 8.2226, Z -8.0000, A 0.000, B 0.000, C 0.000 }
gfCNCPoint5[27115] = {X 401.8551, Y 8.7468, Z -8.0000, A 0.000, B 0.000, C 0.000 }
gfCNCPoint5[27116] = {X 402.5518, Y 9.4435, Z -8.0000, A 0.000, B 0.000, C 0.000 }
gfCNCPoint5[27117] = {X 403.0760, Y 10.2777, Z -8.0000, A 0.000, B 0.000, C 0.000 }
gfCNCPoint5[27118] = {X 403.4014, Y 11.2077, Z -8.0000, A 0.000, B 0.000, C 0.000 }
gfCNCPoint5[27119] = {X 403.5118, Y 12.1868, Z -8.0000, A 0.000, B 0.000, C 0.000 }
gfCNCPoint5[27120] = {X 403.5115, Y 13.0233, Z -8.0000, A 0.000, B 0.000, C 0.000 }
gfCNCPoint5[27121] = {X 403.4070, Y 13.9326, Z -8.0000, A 0.000, B 0.000, C 0.000 }
gfCNCPoint5[27122] = {X 403.1165, Y 14.8007, Z -8.0000, A 0.000, B 0.000, C 0.000 }
gfCNCPoint5[27123] = {X 405.3497, Y 18.6784, Z -8.0000, A 0.000, B 0.000, C 0.000 }
gfCNCPoint5[27124] = {X 407.7804, Y 14.7415, Z -8.0000, A 0.000, B 0.000, C 0.000 }
gfCNCPoint5[27125] = {X 407.5047, Y 13.8788, Z -8.0000, A 0.000, B 0.000, C 0.000 }
gfCNCPoint5[27126] = {X 407.4115, Y 12.9780, Z -8.0000, A 0.000, B 0.000, C 0.000 }
gfCNCPoint5[27127] = {X 407.4115, Y 12.1868, Z -8.0000, A 0.000, B 0.000, C 0.000 }
gfCNCPoint5[27128] = {X 407.5219, Y 11.2077, Z -8.0000, A 0.000, B 0.000, C 0.000 }
gfCNCPoint5[27129] = {X 407.8473, Y 10.2777, Z -8.0000, A 0.000, B 0.000, C 0.000 }
gfCNCPoint5[27130] = {X 408.3715, Y 9.4435, Z -8.0000, A 0.000, B 0.000, C 0.000 }
gfCNCPoint5[27131] = {X 409.0682, Y 8.7468, Z -8.0000, A 0.000, B 0.000, C 0.000 }
gfCNCPoint5[27132] = {X 409.9025, Y 8.2226, Z -8.0000, A 0.000, B 0.000, C 0.000 }
gfCNCPoint5[27133] = {X 410.8324, Y 7.8971, Z -8.0000, A 0.000, B 0.000, C 0.000 }
gfCNCPoint5[27134] = {X 411.8115, Y 7.7868, Z -8.0000, A 0.000, B 0.000, C 0.000 }
gfCNCPoint5[27135] = {X 419.3245, Y 7.7868, Z -8.0000, A 0.000, B 0.000, C 0.000 }
gfCNCPoint5[27136] = {X 420.3036, Y 7.8971, Z -8.0000, A 0.000, B 0.000, C 0.000 }
gfCNCPoint5[27137] = {X 421.2335, Y 8.2226, Z -8.0000, A 0.000, B 0.000, C 0.000 }
gfCNCPoint5[27138] = {X 422.0678, Y 8.7468, Z -8.0000, A 0.000, B 0.000, C 0.000 }
gfCNCPoint5[27139] = {X 422.7645, Y 9.4435, Z -8.0000, A 0.000, B 0.000, C 0.000 }
gfCNCPoint5[27140] = {X 423.2887, Y 10.2777, Z -8.0000, A 0.000, B 0.000, C 0.000 }
gfCNCPoint5[27141] = {X 423.6141, Y 11.2077, Z -8.0000, A 0.000, B 0.000, C 0.000 }
gfCNCPoint5[27142] = {X 423.7245, Y 12.1868, Z -8.0000, A 0.000, B 0.000, C 0.000 }
gfCNCPoint5[27143] = {X 423.7245, Y 12.9806, Z -8.0000, A 0.000, B 0.000, C 0.000 }
gfCNCPoint5[27144] = {X 423.6312, Y 13.8595, Z -8.0000, A 0.000, B 0.000, C 0.000 }
gfCNCPoint5[27145] = {X 423.3665, Y 14.7027, Z -8.0000, A 0.000, B 0.000, C 0.000 }
gfCNCPoint5[27146] = {X 422.9406, Y 15.4772, Z -8.0000, A 0.000, B 0.000, C 0.000 }
gfCNCPoint5[27147] = {X 422.3704, Y 16.1525, Z -8.0000, A 0.000, B 0.000, C 0.000 }
gfCNCPoint5[27148] = {X 421.6782, Y 16.7021, Z -8.0000, A 0.000, B 0.000, C 0.000 }
gfCNCPoint5[27149] = {X 420.8912, Y 17.1044, Z -8.0000, A 0.000, B 0.000, C 0.000 }
gfCNCPoint5[27150] = {X 420.1841, Y 18.0570, Z -8.0000, A 0.000, B 0.000, C 0.000 }
gfCNCPoint5[27151] = {X 419.5441, Y 19.0559, Z -8.0000, A 0.000, B 0.000, C 0.000 }
gfCNCPoint5[27152] = {X 418.0618, Y 21.4551, Z -8.0000, A 0.000, B 0.000, C 0.000 }
gfCNCPoint5[27153] = {X 411.6282, Y 31.7883, Z -8.0000, A 0.000, B 0.000, C 0.000 }
gfCNCPoint5[27154] = {X 411.6288, Y 40.8611, Z -8.0000, A 0.000, B 0.000, C 0.000 }
gfCNCPoint5[27155] = {X 412.2680, Y 41.5580, Z -8.0000, A 0.000, B 0.000, C 0.000 }
gfCNCPoint5[27156] = {X 412.7480, Y 42.3726, Z -8.0000, A 0.000, B 0.000, C 0.000 }
gfCNCPoint5[27157] = {X 413.0480, Y 43.2693, Z -8.0000, A 0.000, B 0.000, C 0.000 }
gfCNCPoint5[27158] = {X 413.1547, Y 44.2088, Z -8.0000, A 0.000, B 0.000, C 0.000 }
gfCNCPoint5[27159] = {X 413.1545, Y 45.0423, Z -8.0000, A 0.000, B 0.000, C 0.000 }
gfCNCPoint5[27160] = {X 413.0719, Y 45.8494, Z -8.0000, A 0.000, B 0.000, C 0.000 }
gfCNCPoint5[27161] = {X 412.8426, Y 46.6276, Z -8.0000, A 0.000, B 0.000, C 0.000 }
gfCNCPoint5[27162] = {X 412.4743, Y 47.3505, Z -8.0000, A 0.000, B 0.000, C 0.000 }
gfCNCPoint5[27163] = {X 411.9795, Y 47.9934, Z -8.0000, A 0.000, B 0.000, C 0.000 }
gfCNCPoint5[27164] = {X 412.3313, Y 48.3200, Z -8.0000, A 0.000, B 0.000, C 0.000 }
gfCNCPoint5[27165] = {X 419.4886, Y 48.3200, Z -8.0000, A 0.000, B 0.000, C 0.000 }
gfCNCPoint5[27166] = {X 420.8006, Y 48.4093, Z -8.0000, A 0.000, B 0.000, C 0.000 }
gfCNCPoint5[27167] = {X 422.0883, Y 48.6756, Z -8.0000, A 0.000, B 0.000, C 0.000 }
gfCNCPoint5[27168] = {X 423.3281, Y 49.1140, Z -8.0000, A 0.000, B 0.000, C 0.000 }
gfCNCPoint5[27169] = {X 424.4970, Y 49.7164, Z -8.0000, A 0.000, B 0.000, C 0.000 }
gfCNCPoint5[27170] = {X 425.4625, Y 50.3832, Z -8.0000, A 0.000, B 0.000, C 0.000 }
gfCNCPoint5[27171] = {X 426.3402, Y 51.1620, Z -8.0000, A 0.000, B 0.000, C 0.000 }
gfCNCPoint5[27172] = {X 427.1172, Y 52.0412, Z -8.0000, A 0.000, B 0.000, C 0.000 }
gfCNCPoint5[27173] = {X 427.7821, Y 53.0080, Z -8.0000, A 0.000, B 0.000, C 0.000 }
gfCNCPoint5[27174] = {X 428.1264, Y 53.6307, Z -8.0000, A 0.000, B 0.000, C 0.000 }
gfCNCPoint5[27175] = {X 428.4240, Y 54.2770, Z -8.0000, A 0.000, B 0.000, C 0.000 }
gfCNCPoint5[27176] = {X 431.5824, Y 55.5075, Z -8.0000, A 0.000, B 0.000, C 0.000 }
gfCNCPoint5[27177] = {X 439.8800, Y 58.7998, Z -8.0000, A 0.000, B 0.000, C 0.000 }
gfCNCPoint5[27178] = {X 441.6502, Y 54.3382, Z -8.0000, A 0.000, B 0.000, C 0.000 }
gfCNCPoint5[27179] = {X 444.2225, Y 55.3588, Z -8.0000, A 0.000, B 0.000, C 0.000 }
gfCNCPoint5[27180] = {X 444.5427, Y 54.0011, Z -8.0000, A 0.000, B 0.000, C 0.000 }
gfCNCPoint5[27181] = {X 444.9921, Y 52.6806, Z -8.0000, A 0.000, B 0.000, C 0.000 }
gfCNCPoint5[27182] = {X 443.9529, Y 53.3760, Z -8.0000, A 0.000, B 0.000, C 0.000 }
gfCNCPoint5[27183] = {X 442.8327, Y 53.9316, Z -8.0000, A 0.000, B 0.000, C 0.000 }
gfCNCPoint5[27184] = {X 441.6502, Y 54.3382, Z -8.0000, A 0.000, B 0.000, C 0.000 }
gfCNCPoint5[27185] = {X 440.7651, Y 56.5690, Z -8.0000, A 0.000, B 0.000, C 0.000 }
gfCNCPoint5[27186] = {X 446.3797, Y 58.7967, Z -8.0000, A 0.000, B 0.000, C 0.000 }
gfCNCPoint5[27187] = {X 446.3796, Y 58.0000, Z -8.0000, A 0.000, B 0.000, C 0.000 }
gfCNCPoint5[27188] = {X 446.4304, Y 56.8936, Z -8.0000, A 0.000, B 0.000, C 0.000 }
gfCNCPoint5[27189] = {X 446.5823, Y 55.7966, Z -8.0000, A 0.000, B 0.000, C 0.000 }
gfCNCPoint5[27190] = {X 446.8494, Y 54.6639, Z -8.0000, A 0.000, B 0.000, C 0.000 }
gfCNCPoint5[27191] = {X 447.2243, Y 53.5622, Z -8.0000, A 0.000, B 0.000, C 0.000 }
gfCNCPoint5[27192] = {X 447.8767, Y 52.1752, Z -8.0000, A 0.000, B 0.000, C 0.000 }
gfCNCPoint5[27193] = {X 448.6995, Y 50.8820, Z -8.0000, A 0.000, B 0.000, C 0.000 }
gfCNCPoint5[27194] = {X 447.8224, Y 50.1272, Z -8.0000, A 0.000, B 0.000, C 0.000 }
gfCNCPoint5[27195] = {X 447.0760, Y 49.2431, Z -8.0000, A 0.000, B 0.000, C 0.000 }
gfCNCPoint5[27196] = {X 446.4792, Y 48.2518, Z -8.0000, A 0.000, B 0.000, C 0.000 }
gfCNCPoint5[27197] = {X 446.0469, Y 47.1785, Z -8.0000, A 0.000, B 0.000, C 0.000 }
gfCNCPoint5[27198] = {X 445.6333, Y 48.2126, Z -8.0000, A 0.000, B 0.000, C 0.000 }
gfCNCPoint5[27199] = {X 445.0668, Y 49.1715, Z -8.0000, A 0.000, B 0.000, C 0.000 }
gfCNCPoint5[27200] = {X 444.3606, Y 50.0328, Z -8.0000, A 0.000, B 0.000, C 0.000 }
gfCNCPoint5[27201] = {X 443.5314, Y 50.7763, Z -8.0000, A 0.000, B 0.000, C 0.000 }
gfCNCPoint5[27202] = {X 442.7498, Y 51.2993, Z -8.0000, A 0.000, B 0.000, C 0.000 }
gfCNCPoint5[27203] = {X 441.9073, Y 51.7171, Z -8.0000, A 0.000, B 0.000, C 0.000 }
gfCNCPoint5[27204] = {X 441.0181, Y 52.0229, Z -8.0000, A 0.000, B 0.000, C 0.000 }
gfCNCPoint5[27205] = {X 440.0678, Y 52.2154, Z -8.0000, A 0.000, B 0.000, C 0.000 }
gfCNCPoint5[27206] = {X 439.1005, Y 52.2800, Z -8.0000, A 0.000, B 0.000, C 0.000 }
gfCNCPoint5[27207] = {X 432.5144, Y 52.2800, Z -8.0000, A 0.000, B 0.000, C 0.000 }
gfCNCPoint5[27208] = {X 431.6034, Y 52.2228, Z -8.0000, A 0.000, B 0.000, C 0.000 }
gfCNCPoint5[27209] = {X 430.7067, Y 52.0520, Z -8.0000, A 0.000, B 0.000, C 0.000 }
gfCNCPoint5[27210] = {X 429.8384, Y 51.7703, Z -8.0000, A 0.000, B 0.000, C 0.000 }
gfCNCPoint5[27211] = {X 430.0166, Y 52.0764, Z -8.0000, A 0.000, B 0.000, C 0.000 }
gfCNCPoint5[27212] = {X 430.1857, Y 52.3876, Z -8.0000, A 0.000, B 0.000, C 0.000 }
gfCNCPoint5[27213] = {X 432.4641, Y 53.2753, Z -8.0000, A 0.000, B 0.000, C 0.000 }
gfCNCPoint5[27214] = {X 440.7651, Y 56.5690, Z -8.0000, A 0.000, B 0.000, C 0.000 }
gfCNCPoint5[27215] = {X 439.8800, Y 58.7998, Z -8.0000, A 0.000, B 0.000, C 0.000 }
gfCNCPoint5[27216] = {X 449.5090, Y 62.6204, Z -8.0000, A 0.000, B 0.000, C 0.000 }
gfCNCPoint5[27217] = {X 449.1111, Y 61.4458, Z -8.0000, A 0.000, B 0.000, C 0.000 }
gfCNCPoint5[27218] = {X 448.8667, Y 60.2300, Z -8.0000, A 0.000, B 0.000, C 0.000 }
gfCNCPoint5[27219] = {X 448.7798, Y 58.9930, Z -8.0000, A 0.000, B 0.000, C 0.000 }
gfCNCPoint5[27220] = {X 448.7796, Y 58.0000, Z -8.0000, A 0.000, B 0.000, C 0.000 }
gfCNCPoint5[27221] = {X 448.8564, Y 56.7833, Z -8.0000, A 0.000, B 0.000, C 0.000 }
gfCNCPoint5[27222] = {X 449.0855, Y 55.5859, Z -8.0000, A 0.000, B 0.000, C 0.000 }
gfCNCPoint5[27223] = {X 449.4632, Y 54.4268, Z -8.0000, A 0.000, B 0.000, C 0.000 }
gfCNCPoint5[27224] = {X 449.9837, Y 53.3244, Z -8.0000, A 0.000, B 0.000, C 0.000 }
gfCNCPoint5[27225] = {X 450.6386, Y 52.2961, Z -8.0000, A 0.000, B 0.000, C 0.000 }
gfCNCPoint5[27226] = {X 451.3887, Y 51.3890, Z -8.0000, A 0.000, B 0.000, C 0.000 }
gfCNCPoint5[27227] = {X 452.2434, Y 50.5796, Z -8.0000, A 0.000, B 0.000, C 0.000 }
gfCNCPoint5[27228] = {X 453.1901, Y 49.8800, Z -8.0000, A 0.000, B 0.000, C 0.000 }
gfCNCPoint5[27229] = {X 452.3731, Y 49.8442, Z -8.0000, A 0.000, B 0.000, C 0.000 }
gfCNCPoint5[27230] = {X 451.5735, Y 49.6724, Z -8.0000, A 0.000, B 0.000, C 0.000 }
gfCNCPoint5[27231] = {X 450.8138, Y 49.3696, Z -8.0000, A 0.000, B 0.000, C 0.000 }
gfCNCPoint5[27232] = {X 450.1154, Y 48.9441, Z -8.0000, A 0.000, B 0.000, C 0.000 }
gfCNCPoint5[27233] = {X 449.3503, Y 48.2496, Z -8.0000, A 0.000, B 0.000, C 0.000 }
gfCNCPoint5[27234] = {X 448.7486, Y 47.4095, Z -8.0000, A 0.000, B 0.000, C 0.000 }
gfCNCPoint5[27235] = {X 448.3373, Y 46.4616, Z -8.0000, A 0.000, B 0.000, C 0.000 }
gfCNCPoint5[27236] = {X 448.1732, Y 45.7588, Z -8.0000, A 0.000, B 0.000, C 0.000 }
gfCNCPoint5[27237] = {X 448.1146, Y 45.0395, Z -8.0000, A 0.000, B 0.000, C 0.000 }
gfCNCPoint5[27238] = {X 448.1149, Y 44.1416, Z -8.0000, A 0.000, B 0.000, C 0.000 }
gfCNCPoint5[27239] = {X 448.2252, Y 43.1751, Z -8.0000, A 0.000, B 0.000, C 0.000 }
gfCNCPoint5[27240] = {X 448.5250, Y 42.2496, Z -8.0000, A 0.000, B 0.000, C 0.000 }
gfCNCPoint5[27241] = {X 449.0024, Y 41.4020, Z -8.0000, A 0.000, B 0.000, C 0.000 }
gfCNCPoint5[27242] = {X 449.6384, Y 40.6660, Z -8.0000, A 0.000, B 0.000, C 0.000 }
gfCNCPoint5[27243] = {X 449.6384, Y 35.0338, Z -8.0000, A 0.000, B 0.000, C 0.000 }
gfCNCPoint5[27244] = {X 447.8176, Y 35.0338, Z -8.0000, A 0.000, B 0.000, C 0.000 }
gfCNCPoint5[27245] = {X 443.7932, Y 42.8699, Z -8.0000, A 0.000, B 0.000, C 0.000 }
gfCNCPoint5[27246] = {X 443.9304, Y 43.5113, Z -8.0000, A 0.000, B 0.000, C 0.000 }
gfCNCPoint5[27247] = {X 443.9803, Y 44.1653, Z -8.0000, A 0.000, B 0.000, C 0.000 }
gfCNCPoint5[27248] = {X 443.9805, Y 45.0000, Z -8.0000, A 0.000, B 0.000, C 0.000 }
gfCNCPoint5[27249] = {X 443.9242, Y 45.7387, Z -8.0000, A 0.000, B 0.000, C 0.000 }
gfCNCPoint5[27250] = {X 443.7568, Y 46.4603, Z -8.0000, A 0.000, B 0.000, C 0.000 }
gfCNCPoint5[27251] = {X 443.3474, Y 47.4038, Z -8.0000, A 0.000, B 0.000, C 0.000 }
gfCNCPoint5[27252] = {X 442.7493, Y 48.2405, Z -8.0000, A 0.000, B 0.000, C 0.000 }
gfCNCPoint5[27253] = {X 441.9891, Y 48.9332, Z -8.0000, A 0.000, B 0.000, C 0.000 }
gfCNCPoint5[27254] = {X 441.1006, Y 49.4513, Z -8.0000, A 0.000, B 0.000, C 0.000 }
gfCNCPoint5[27255] = {X 440.1232, Y 49.7716, Z -8.0000, A 0.000, B 0.000, C 0.000 }
gfCNCPoint5[27256] = {X 439.1005, Y 49.8800, Z -8.0000, A 0.000, B 0.000, C 0.000 }
gfCNCPoint5[27257] = {X 432.5144, Y 49.8800, Z -8.0000, A 0.000, B 0.000, C 0.000 }
gfCNCPoint5[27258] = {X 431.6014, Y 49.7938, Z -8.0000, A 0.000, B 0.000, C 0.000 }
gfCNCPoint5[27259] = {X 430.7206, Y 49.5383, Z -8.0000, A 0.000, B 0.000, C 0.000 }
gfCNCPoint5[27260] = {X 429.8343, Y 49.0782, Z -8.0000, A 0.000, B 0.000, C 0.000 }
gfCNCPoint5[27261] = {X 429.0603, Y 48.4473, Z -8.0000, A 0.000, B 0.000, C 0.000 }
gfCNCPoint5[27262] = {X 428.4309, Y 47.6720, Z -8.0000, A 0.000, B 0.000, C 0.000 }
gfCNCPoint5[27263] = {X 427.9725, Y 46.7848, Z -8.0000, A 0.000, B 0.000, C 0.000 }
gfCNCPoint5[27264] = {X 427.7197, Y 45.9083, Z -8.0000, A 0.000, B 0.000, C 0.000 }
gfCNCPoint5[27265] = {X 427.6344, Y 45.0000, Z -8.0000, A 0.000, B 0.000, C 0.000 }
gfCNCPoint5[27266] = {X 427.6344, Y 44.2089, Z -8.0000, A 0.000, B 0.000, C 0.000 }
gfCNCPoint5[27267] = {X 427.7263, Y 43.2661, Z -8.0000, A 0.000, B 0.000, C 0.000 }
gfCNCPoint5[27268] = {X 427.9987, Y 42.3588, Z -8.0000, A 0.000, B 0.000, C 0.000 }
gfCNCPoint5[27269] = {X 428.4412, Y 41.5212, Z -8.0000, A 0.000, B 0.000, C 0.000 }
gfCNCPoint5[27270] = {X 429.0371, Y 40.7849, Z -8.0000, A 0.000, B 0.000, C 0.000 }
gfCNCPoint5[27271] = {X 429.7641, Y 40.1776, Z -8.0000, A 0.000, B 0.000, C 0.000 }
gfCNCPoint5[27272] = {X 430.5947, Y 39.7222, Z -8.0000, A 0.000, B 0.000, C 0.000 }
gfCNCPoint5[27273] = {X 434.2528, Y 32.5619, Z -8.0000, A 0.000, B 0.000, C 0.000 }
gfCNCPoint5[27274] = {X 432.9259, Y 31.5655, Z -8.0000, A 0.000, B 0.000, C 0.000 }
gfCNCPoint5[27275] = {X 431.7506, Y 30.3940, Z -8.0000, A 0.000, B 0.000, C 0.000 }
gfCNCPoint5[27276] = {X 430.7498, Y 29.0703, Z -8.0000, A 0.000, B 0.000, C 0.000 }
gfCNCPoint5[27277] = {X 429.9430, Y 27.6203, Z -8.0000, A 0.000, B 0.000, C 0.000 }
gfCNCPoint5[27278] = {X 429.3458, Y 26.0720, Z -8.0000, A 0.000, B 0.000, C 0.000 }
gfCNCPoint5[27279] = {X 428.8987, Y 24.1619, Z -8.0000, A 0.000, B 0.000, C 0.000 }
gfCNCPoint5[27280] = {X 428.6733, Y 22.2131, Z -8.0000, A 0.000, B 0.000, C 0.000 }
gfCNCPoint5[27281] = {X 428.6727, Y 20.2514, Z -8.0000, A 0.000, B 0.000, C 0.000 }
gfCNCPoint5[27282] = {X 428.8969, Y 18.3025, Z -8.0000, A 0.000, B 0.000, C 0.000 }
gfCNCPoint5[27283] = {X 429.3429, Y 16.3921, Z -8.0000, A 0.000, B 0.000, C 0.000 }
gfCNCPoint5[27284] = {X 429.8636, Y 14.9597, Z -8.0000, A 0.000, B 0.000, C 0.000 }
gfCNCPoint5[27285] = {X 430.5563, Y 13.6021, Z -8.0000, A 0.000, B 0.000, C 0.000 }
gfCNCPoint5[27286] = {X 431.4104, Y 12.3397, Z -8.0000, A 0.000, B 0.000, C 0.000 }
gfCNCPoint5[27287] = {X 432.4130, Y 11.1918, Z -8.0000, A 0.000, B 0.000, C 0.000 }
gfCNCPoint5[27288] = {X 433.5446, Y 10.1791, Z -8.0000, A 0.000, B 0.000, C 0.000 }
gfCNCPoint5[27289] = {X 434.7916, Y 9.3125, Z -8.0000, A 0.000, B 0.000, C 0.000 }
gfCNCPoint5[27290] = {X 436.1353, Y 8.6049, Z -8.0000, A 0.000, B 0.000, C 0.000 }
gfCNCPoint5[27291] = {X 437.5555, Y 8.0671, Z -8.0000, A 0.000, B 0.000, C 0.000 }
gfCNCPoint5[27292] = {X 439.0307, Y 7.7070, Z -8.0000, A 0.000, B 0.000, C 0.000 }
gfCNCPoint5[27293] = {X 441.1775, Y 7.4098, Z -8.0000, A 0.000, B 0.000, C 0.000 }
gfCNCPoint5[27294] = {X 443.3425, Y 7.3133, Z -8.0000, A 0.000, B 0.000, C 0.000 }
gfCNCPoint5[27295] = {X 444.0315, Y 7.3092, Z -8.0000, A 0.000, B 0.000, C 0.000 }
gfCNCPoint5[27296] = {X 459.4469, Y 7.3092, Z -8.0000, A 0.000, B 0.000, C 0.000 }
gfCNCPoint5[27297] = {X 460.4098, Y 7.4054, Z -8.0000, A 0.000, B 0.000, C 0.000 }
gfCNCPoint5[27298] = {X 461.3348, Y 7.6900, Z -8.0000, A 0.000, B 0.000, C 0.000 }
gfCNCPoint5[27299] = {X 462.1852, Y 8.1518, Z -8.0000, A 0.000, B 0.000, C 0.000 }
gfCNCPoint5[27300] = {X 462.9275, Y 8.7726, Z -8.0000, A 0.000, B 0.000, C 0.000 }
gfCNCPoint5[27301] = {X 463.5325, Y 9.5279, Z -8.0000, A 0.000, B 0.000, C 0.000 }
gfCNCPoint5[27302] = {X 463.9762, Y 10.3879, Z -8.0000, A 0.000, B 0.000, C 0.000 }
gfCNCPoint5[27303] = {X 464.2317, Y 11.2680, Z -8.0000, A 0.000, B 0.000, C 0.000 }
gfCNCPoint5[27304] = {X 464.3179, Y 12.1803, Z -8.0000, A 0.000, B 0.000, C 0.000 }
gfCNCPoint5[27305] = {X 464.3179, Y 12.9780, Z -8.0000, A 0.000, B 0.000, C 0.000 }
gfCNCPoint5[27306] = {X 464.2175, Y 13.9632, Z -8.0000, A 0.000, B 0.000, C 0.000 }
gfCNCPoint5[27307] = {X 463.9201, Y 14.9079, Z -8.0000, A 0.000, B 0.000, C 0.000 }
gfCNCPoint5[27308] = {X 463.4382, Y 15.7731, Z -8.0000, A 0.000, B 0.000, C 0.000 }
gfCNCPoint5[27309] = {X 462.7915, Y 16.5231, Z -8.0000, A 0.000, B 0.000, C 0.000 }
gfCNCPoint5[27310] = {X 462.7913, Y 16.7695, Z -8.0000, A 0.000, B 0.000, C 0.000 }
gfCNCPoint5[27311] = {X 462.7917, Y 25.8898, Z -8.0000, A 0.000, B 0.000, C 0.000 }
gfCNCPoint5[27312] = {X 467.5917, Y 25.8896, Z -8.0000, A 0.000, B 0.000, C 0.000 }
gfCNCPoint5[27313] = {X 467.5922, Y 38.9924, Z -8.0000, A 0.000, B 0.000, C 0.000 }
gfCNCPoint5[27314] = {X 467.6015, Y 39.0069, Z -8.0000, A 0.000, B 0.000, C 0.000 }
gfCNCPoint5[27315] = {X 468.3506, Y 37.9855, Z -8.0000, A 0.000, B 0.000, C 0.000 }
gfCNCPoint5[27316] = {X 469.2267, Y 37.0706, Z -8.0000, A 0.000, B 0.000, C 0.000 }
gfCNCPoint5[27317] = {X 470.2148, Y 36.2780, Z -8.0000, A 0.000, B 0.000, C 0.000 }
gfCNCPoint5[27318] = {X 471.5268, Y 33.7098, Z -8.0000, A 0.000, B 0.000, C 0.000 }
gfCNCPoint5[27319] = {X 470.4791, Y 32.4133, Z -8.0000, A 0.000, B 0.000, C 0.000 }
gfCNCPoint5[27320] = {X 469.5649, Y 31.0194, Z -8.0000, A 0.000, B 0.000, C 0.000 }
gfCNCPoint5[27321] = {X 468.7932, Y 29.5419, Z -8.0000, A 0.000, B 0.000, C 0.000 }
gfCNCPoint5[27322] = {X 468.1717, Y 27.9951, Z -8.0000, A 0.000, B 0.000, C 0.000 }
gfCNCPoint5[27323] = {X 467.7063, Y 26.3945, Z -8.0000, A 0.000, B 0.000, C 0.000 }
gfCNCPoint5[27324] = {X 467.6475, Y 26.1423, Z -8.0000, A 0.000, B 0.000, C 0.000 }
gfCNCPoint5[27325] = {X 467.5917, Y 25.8896, Z -8.0000, A 0.000, B 0.000, C 0.000 }
gfCNCPoint5[27326] = {X 465.1917, Y 25.8897, Z -8.0000, A 0.000, B 0.000, C 0.000 }
gfCNCPoint5[27327] = {X 465.1922, Y 39.7493, Z -8.0000, A 0.000, B 0.000, C 0.000 }
gfCNCPoint5[27328] = {X 465.3911, Y 40.0186, Z -8.0000, A 0.000, B 0.000, C 0.000 }
gfCNCPoint5[27329] = {X 465.5774, Y 40.2966, Z -8.0000, A 0.000, B 0.000, C 0.000 }
gfCNCPoint5[27330] = {X 466.0634, Y 41.1919, Z -8.0000, A 0.000, B 0.000, C 0.000 }
gfCNCPoint5[27331] = {X 466.4196, Y 42.1462, Z -8.0000, A 0.000, B 0.000, C 0.000 }
gfCNCPoint5[27332] = {X 466.6392, Y 43.1408, Z -8.0000, A 0.000, B 0.000, C 0.000 }
gfCNCPoint5[27333] = {X 466.7178, Y 44.1564, Z -8.0000, A 0.000, B 0.000, C 0.000 }
gfCNCPoint5[27334] = {X 466.7179, Y 45.0000, Z -8.0000, A 0.000, B 0.000, C 0.000 }
gfCNCPoint5[27335] = {X 466.7033, Y 45.4609, Z -8.0000, A 0.000, B 0.000, C 0.000 }
gfCNCPoint5[27336] = {X 466.6596, Y 45.9200, Z -8.0000, A 0.000, B 0.000, C 0.000 }
gfCNCPoint5[27337] = {X 468.5433, Y 45.9200, Z -8.0000, A 0.000, B 0.000, C 0.000 }
gfCNCPoint5[27338] = {X 468.4996, Y 45.4609, Z -8.0000, A 0.000, B 0.000, C 0.000 }
gfCNCPoint5[27339] = {X 468.4850, Y 45.0000, Z -8.0000, A 0.000, B 0.000, C 0.000 }
gfCNCPoint5[27340] = {X 468.4850, Y 44.2089, Z -8.0000, A 0.000, B 0.000, C 0.000 }
gfCNCPoint5[27341] = {X 468.5581, Y 43.1798, Z -8.0000, A 0.000, B 0.000, C 0.000 }
gfCNCPoint5[27342] = {X 468.7759, Y 42.1713, Z -8.0000, A 0.000, B 0.000, C 0.000 }
gfCNCPoint5[27343] = {X 469.1341, Y 41.2038, Z -8.0000, A 0.000, B 0.000, C 0.000 }
gfCNCPoint5[27344] = {X 469.6255, Y 40.2966, Z -8.0000, A 0.000, B 0.000, C 0.000 }
gfCNCPoint5[27345] = {X 470.3102, Y 39.3876, Z -8.0000, A 0.000, B 0.000, C 0.000 }
gfCNCPoint5[27346] = {X 471.1282, Y 38.5964, Z -8.0000, A 0.000, B 0.000, C 0.000 }
gfCNCPoint5[27347] = {X 472.0595, Y 37.9424, Z -8.0000, A 0.000, B 0.000, C 0.000 }
gfCNCPoint5[27348] = {X 474.4563, Y 33.2510, Z -8.0000, A 0.000, B 0.000, C 0.000 }
gfCNCPoint5[27349] = {X 473.2240, Y 32.0063, Z -8.0000, A 0.000, B 0.000, C 0.000 }
gfCNCPoint5[27350] = {X 472.1518, Y 30.6213, Z -8.0000, A 0.000, B 0.000, C 0.000 }
gfCNCPoint5[27351] = {X 471.2555, Y 29.1164, Z -8.0000, A 0.000, B 0.000, C 0.000 }
gfCNCPoint5[27352] = {X 470.5484, Y 27.5140, Z -8.0000, A 0.000, B 0.000, C 0.000 }
gfCNCPoint5[27353] = {X 470.0408, Y 25.8376, Z -8.0000, A 0.000, B 0.000, C 0.000 }
gfCNCPoint5[27354] = {X 469.9882, Y 25.6119, Z -8.0000, A 0.000, B 0.000, C 0.000 }
gfCNCPoint5[27355] = {X 469.9381, Y 25.3855, Z -8.0000, A 0.000, B 0.000, C 0.000 }
gfCNCPoint5[27356] = {X 469.6266, Y 23.4897, Z -8.0000, A 0.000, B 0.000, C 0.000 }
gfCNCPoint5[27357] = {X 469.5011, Y 21.5726, Z -8.0000, A 0.000, B 0.000, C 0.000 }
gfCNCPoint5[27358] = {X 469.5628, Y 19.6524, Z -8.0000, A 0.000, B 0.000, C 0.000 }
gfCNCPoint5[27359] = {X 469.8111, Y 17.7473, Z -8.0000, A 0.000, B 0.000, C 0.000 }
gfCNCPoint5[27360] = {X 470.2437, Y 15.8754, Z -8.0000, A 0.000, B 0.000, C 0.000 }
gfCNCPoint5[27361] = {X 470.6906, Y 14.5429, Z -8.0000, A 0.000, B 0.000, C 0.000 }
gfCNCPoint5[27362] = {X 471.2619, Y 13.2588, Z -8.0000, A 0.000, B 0.000, C 0.000 }
gfCNCPoint5[27363] = {X 469.1179, Y 12.1802, Z -8.0000, A 0.000, B 0.000, C 0.000 }
gfCNCPoint5[27364] = {X 469.1881, Y 12.0422, Z -8.0000, A 0.000, B 0.000, C 0.000 }
gfCNCPoint5[27365] = {X 469.2596, Y 11.9048, Z -8.0000, A 0.000, B 0.000, C 0.000 }
gfCNCPoint5[27366] = {X 469.1140, Y 11.9048, Z -8.0000, A 0.000, B 0.000, C 0.000 }
gfCNCPoint5[27367] = {X 469.1170, Y 12.0425, Z -8.0000, A 0.000, B 0.000, C 0.000 }
gfCNCPoint5[27368] = {X 469.1179, Y 12.1802, Z -8.0000, A 0.000, B 0.000, C 0.000 }
gfCNCPoint5[27369] = {X 471.2619, Y 13.2588, Z -8.0000, A 0.000, B 0.000, C 0.000 }
gfCNCPoint5[27370] = {X 471.3223, Y 13.1401, Z -8.0000, A 0.000, B 0.000, C 0.000 }
gfCNCPoint5[27371] = {X 471.3838, Y 13.0219, Z -8.0000, A 0.000, B 0.000, C 0.000 }
gfCNCPoint5[27372] = {X 472.1250, Y 11.7667, Z -8.0000, A 0.000, B 0.000, C 0.000 }
gfCNCPoint5[27373] = {X 472.9861, Y 10.5905, Z -8.0000, A 0.000, B 0.000, C 0.000 }
gfCNCPoint5[27374] = {X 473.9588, Y 9.5048, Z -8.0000, A 0.000, B 0.000, C 0.000 }
gfCNCPoint5[27375] = {X 466.2078, Y 9.5048, Z -8.0000, A 0.000, B 0.000, C 0.000 }
gfCNCPoint5[27376] = {X 466.5692, Y 10.7169, Z -8.0000, A 0.000, B 0.000, C 0.000 }
gfCNCPoint5[27377] = {X 466.7150, Y 11.9732, Z -8.0000, A 0.000, B 0.000, C 0.000 }
gfCNCPoint5[27378] = {X 466.7172, Y 12.0767, Z -8.0000, A 0.000, B 0.000, C 0.000 }
gfCNCPoint5[27379] = {X 466.7179, Y 12.1803, Z -8.0000, A 0.000, B 0.000, C 0.000 }
gfCNCPoint5[27380] = {X 466.7179, Y 12.9780, Z -8.0000, A 0.000, B 0.000, C 0.000 }
gfCNCPoint5[27381] = {X 466.6192, Y 14.1728, Z -8.0000, A 0.000, B 0.000, C 0.000 }
gfCNCPoint5[27382] = {X 466.3257, Y 15.3353, Z -8.0000, A 0.000, B 0.000, C 0.000 }
gfCNCPoint5[27383] = {X 465.8454, Y 16.4338, Z -8.0000, A 0.000, B 0.000, C 0.000 }
gfCNCPoint5[27384] = {X 465.1913, Y 17.4386, Z -8.0000, A 0.000, B 0.000, C 0.000 }
gfCNCPoint5[27385] = {X 465.1917, Y 25.8897, Z -8.0000, A 0.000, B 0.000, C 0.000 }
gfCNCPoint5[27386] = {X 462.7917, Y 25.8898, Z -8.0000, A 0.000, B 0.000, C 0.000 }
gfCNCPoint5[27387] = {X 462.7922, Y 40.6644, Z -8.0000, A 0.000, B 0.000, C 0.000 }
gfCNCPoint5[27388] = {X 463.4326, Y 41.4058, Z -8.0000, A 0.000, B 0.000, C 0.000 }
gfCNCPoint5[27389] = {X 463.9120, Y 42.2602, Z -8.0000, A 0.000, B 0.000, C 0.000 }
gfCNCPoint5[27390] = {X 464.2111, Y 43.1931, Z -8.0000, A 0.000, B 0.000, C 0.000 }
gfCNCPoint5[27391] = {X 464.3178, Y 44.1670, Z -8.0000, A 0.000, B 0.000, C 0.000 }
gfCNCPoint5[27392] = {X 464.3179, Y 45.0000, Z -8.0000, A 0.000, B 0.000, C 0.000 }
gfCNCPoint5[27393] = {X 464.3082, Y 45.3090, Z -8.0000, A 0.000, B 0.000, C 0.000 }
gfCNCPoint5[27394] = {X 464.2788, Y 45.6167, Z -8.0000, A 0.000, B 0.000, C 0.000 }
gfCNCPoint5[27395] = {X 464.0485, Y 46.5992, Z -8.0000, A 0.000, B 0.000, C 0.000 }
gfCNCPoint5[27396] = {X 463.6209, Y 47.5134, Z -8.0000, A 0.000, B 0.000, C 0.000 }
gfCNCPoint5[27397] = {X 463.0145, Y 48.3200, Z -8.0000, A 0.000, B 0.000, C 0.000 }
gfCNCPoint5[27398] = {X 462.6627, Y 47.9934, Z -8.0000, A 0.000, B 0.000, C 0.000 }
gfCNCPoint5[27399] = {X 461.9835, Y 48.5889, Z -8.0000, A 0.000, B 0.000, C 0.000 }
gfCNCPoint5[27400] = {X 461.1970, Y 49.0331, Z -8.0000, A 0.000, B 0.000, C 0.000 }
gfCNCPoint5[27401] = {X 460.3364, Y 49.3073, Z -8.0000, A 0.000, B 0.000, C 0.000 }
gfCNCPoint5[27402] = {X 459.4379, Y 49.4000, Z -8.0000, A 0.000, B 0.000, C 0.000 }
gfCNCPoint5[27403] = {X 452.9945, Y 49.4000, Z -8.0000, A 0.000, B 0.000, C 0.000 }
gfCNCPoint5[27404] = {X 452.0154, Y 49.2897, Z -8.0000, A 0.000, B 0.000, C 0.000 }
gfCNCPoint5[27405] = {X 451.0854, Y 48.9643, Z -8.0000, A 0.000, B 0.000, C 0.000 }
gfCNCPoint5[27406] = {X 450.2511, Y 48.4401, Z -8.0000, A 0.000, B 0.000, C 0.000 }
gfCNCPoint5[27407] = {X 449.5544, Y 47.7433, Z -8.0000, A 0.000, B 0.000, C 0.000 }
gfCNCPoint5[27408] = {X 449.0302, Y 46.9091, Z -8.0000, A 0.000, B 0.000, C 0.000 }
gfCNCPoint5[27409] = {X 448.7048, Y 45.9791, Z -8.0000, A 0.000, B 0.000, C 0.000 }
gfCNCPoint5[27410] = {X 448.5945, Y 45.0000, Z -8.0000, A 0.000, B 0.000, C 0.000 }
gfCNCPoint5[27411] = {X 448.5949, Y 44.1483, Z -8.0000, A 0.000, B 0.000, C 0.000 }
gfCNCPoint5[27412] = {X 448.7053, Y 43.2275, Z -8.0000, A 0.000, B 0.000, C 0.000 }
gfCNCPoint5[27413] = {X 449.0063, Y 42.3503, Z -8.0000, A 0.000, B 0.000, C 0.000 }
gfCNCPoint5[27414] = {X 449.4844, Y 41.5556, Z -8.0000, A 0.000, B 0.000, C 0.000 }
gfCNCPoint5[27415] = {X 450.1184, Y 40.8789, Z -8.0000, A 0.000, B 0.000, C 0.000 }
gfCNCPoint5[27416] = {X 450.1184, Y 34.5538, Z -8.0000, A 0.000, B 0.000, C 0.000 }
gfCNCPoint5[27417] = {X 447.5245, Y 34.5538, Z -8.0000, A 0.000, B 0.000, C 0.000 }
gfCNCPoint5[27418] = {X 443.2770, Y 42.8244, Z -8.0000, A 0.000, B 0.000, C 0.000 }
gfCNCPoint5[27419] = {X 443.4442, Y 43.5077, Z -8.0000, A 0.000, B 0.000, C 0.000 }
gfCNCPoint5[27420] = {X 443.5005, Y 44.2089, Z -8.0000, A 0.000, B 0.000, C 0.000 }
gfCNCPoint5[27421] = {X 443.5005, Y 45.0000, Z -8.0000, A 0.000, B 0.000, C 0.000 }
gfCNCPoint5[27422] = {X 443.3902, Y 45.9791, Z -8.0000, A 0.000, B 0.000, C 0.000 }
gfCNCPoint5[27423] = {X 443.0647, Y 46.9091, Z -8.0000, A 0.000, B 0.000, C 0.000 }
gfCNCPoint5[27424] = {X 442.5405, Y 47.7434, Z -8.0000, A 0.000, B 0.000, C 0.000 }
gfCNCPoint5[27425] = {X 441.8438, Y 48.4401, Z -8.0000, A 0.000, B 0.000, C 0.000 }
gfCNCPoint5[27426] = {X 441.0096, Y 48.9643, Z -8.0000, A 0.000, B 0.000, C 0.000 }
gfCNCPoint5[27427] = {X 440.0796, Y 49.2897, Z -8.0000, A 0.000, B 0.000, C 0.000 }
gfCNCPoint5[27428] = {X 439.1005, Y 49.4000, Z -8.0000, A 0.000, B 0.000, C 0.000 }
gfCNCPoint5[27429] = {X 432.5144, Y 49.4000, Z -8.0000, A 0.000, B 0.000, C 0.000 }
gfCNCPoint5[27430] = {X 431.5353, Y 49.2897, Z -8.0000, A 0.000, B 0.000, C 0.000 }
gfCNCPoint5[27431] = {X 430.6053, Y 48.9643, Z -8.0000, A 0.000, B 0.000, C 0.000 }
gfCNCPoint5[27432] = {X 429.7711, Y 48.4401, Z -8.0000, A 0.000, B 0.000, C 0.000 }
gfCNCPoint5[27433] = {X 429.0743, Y 47.7434, Z -8.0000, A 0.000, B 0.000, C 0.000 }
gfCNCPoint5[27434] = {X 428.5501, Y 46.9091, Z -8.0000, A 0.000, B 0.000, C 0.000 }
gfCNCPoint5[27435] = {X 428.2247, Y 45.9791, Z -8.0000, A 0.000, B 0.000, C 0.000 }
gfCNCPoint5[27436] = {X 428.1144, Y 45.0000, Z -8.0000, A 0.000, B 0.000, C 0.000 }
gfCNCPoint5[27437] = {X 428.1148, Y 44.1483, Z -8.0000, A 0.000, B 0.000, C 0.000 }
gfCNCPoint5[27438] = {X 428.2132, Y 43.2816, Z -8.0000, A 0.000, B 0.000, C 0.000 }
gfCNCPoint5[27439] = {X 428.4806, Y 42.4514, Z -8.0000, A 0.000, B 0.000, C 0.000 }
gfCNCPoint5[27440] = {X 428.9065, Y 41.6903, Z -8.0000, A 0.000, B 0.000, C 0.000 }
gfCNCPoint5[27441] = {X 429.4741, Y 41.0281, Z -8.0000, A 0.000, B 0.000, C 0.000 }
gfCNCPoint5[27442] = {X 430.1613, Y 40.4909, Z -8.0000, A 0.000, B 0.000, C 0.000 }
gfCNCPoint5[27443] = {X 430.9408, Y 40.0998, Z -8.0000, A 0.000, B 0.000, C 0.000 }
gfCNCPoint5[27444] = {X 434.8812, Y 32.3870, Z -8.0000, A 0.000, B 0.000, C 0.000 }
gfCNCPoint5[27445] = {X 433.7238, Y 31.5991, Z -8.0000, A 0.000, B 0.000, C 0.000 }
gfCNCPoint5[27446] = {X 432.6717, Y 30.6753, Z -8.0000, A 0.000, B 0.000, C 0.000 }
gfCNCPoint5[27447] = {X 431.7406, Y 29.6297, Z -8.0000, A 0.000, B 0.000, C 0.000 }
gfCNCPoint5[27448] = {X 430.9446, Y 28.4779, Z -8.0000, A 0.000, B 0.000, C 0.000 }
gfCNCPoint5[27449] = {X 430.2955, Y 27.2373, Z -8.0000, A 0.000, B 0.000, C 0.000 }
gfCNCPoint5[27450] = {X 429.8033, Y 25.9265, Z -8.0000, A 0.000, B 0.000, C 0.000 }
gfCNCPoint5[27451] = {X 429.3702, Y 24.0718, Z -8.0000, A 0.000, B 0.000, C 0.000 }
gfCNCPoint5[27452] = {X 429.1521, Y 22.1796, Z -8.0000, A 0.000, B 0.000, C 0.000 }
gfCNCPoint5[27453] = {X 429.1521, Y 20.2749, Z -8.0000, A 0.000, B 0.000, C 0.000 }
gfCNCPoint5[27454] = {X 429.3702, Y 18.3827, Z -8.0000, A 0.000, B 0.000, C 0.000 }
gfCNCPoint5[27455] = {X 429.8033, Y 16.5279, Z -8.0000, A 0.000, B 0.000, C 0.000 }
gfCNCPoint5[27456] = {X 430.3769, Y 14.9864, Z -8.0000, A 0.000, B 0.000, C 0.000 }
gfCNCPoint5[27457] = {X 431.1575, Y 13.5386, Z -8.0000, A 0.000, B 0.000, C 0.000 }
gfCNCPoint5[27458] = {X 432.1300, Y 12.2122, Z -8.0000, A 0.000, B 0.000, C 0.000 }
gfCNCPoint5[27459] = {X 433.2760, Y 11.0324, Z -8.0000, A 0.000, B 0.000, C 0.000 }
gfCNCPoint5[27460] = {X 434.5737, Y 10.0217, Z -8.0000, A 0.000, B 0.000, C 0.000 }
gfCNCPoint5[27461] = {X 435.9982, Y 9.1995, Z -8.0000, A 0.000, B 0.000, C 0.000 }
gfCNCPoint5[27462] = {X 437.5224, Y 8.5814, Z -8.0000, A 0.000, B 0.000, C 0.000 }
gfCNCPoint5[27463] = {X 439.1172, Y 8.1791, Z -8.0000, A 0.000, B 0.000, C 0.000 }
gfCNCPoint5[27464] = {X 441.2213, Y 7.8878, Z -8.0000, A 0.000, B 0.000, C 0.000 }
gfCNCPoint5[27465] = {X 443.3434, Y 7.7933, Z -8.0000, A 0.000, B 0.000, C 0.000 }
gfCNCPoint5[27466] = {X 444.0367, Y 7.7892, Z -8.0000, A 0.000, B 0.000, C 0.000 }
gfCNCPoint5[27467] = {X 459.4469, Y 7.7892, Z -8.0000, A 0.000, B 0.000, C 0.000 }
gfCNCPoint5[27468] = {X 460.4240, Y 7.8993, Z -8.0000, A 0.000, B 0.000, C 0.000 }
gfCNCPoint5[27469] = {X 461.3521, Y 8.2241, Z -8.0000, A 0.000, B 0.000, C 0.000 }
gfCNCPoint5[27470] = {X 462.1847, Y 8.7472, Z -8.0000, A 0.000, B 0.000, C 0.000 }
gfCNCPoint5[27471] = {X 462.8800, Y 9.4425, Z -8.0000, A 0.000, B 0.000, C 0.000 }
gfCNCPoint5[27472] = {X 463.4031, Y 10.2751, Z -8.0000, A 0.000, B 0.000, C 0.000 }
gfCNCPoint5[27473] = {X 463.7278, Y 11.2032, Z -8.0000, A 0.000, B 0.000, C 0.000 }
gfCNCPoint5[27474] = {X 463.8379, Y 12.1803, Z -8.0000, A 0.000, B 0.000, C 0.000 }
gfCNCPoint5[27475] = {X 463.8377, Y 13.0201, Z -8.0000, A 0.000, B 0.000, C 0.000 }
gfCNCPoint5[27476] = {X 463.7300, Y 13.9466, Z -8.0000, A 0.000, B 0.000, C 0.000 }
gfCNCPoint5[27477] = {X 463.4294, Y 14.8295, Z -8.0000, A 0.000, B 0.000, C 0.000 }
gfCNCPoint5[27478] = {X 462.9495, Y 15.6293, Z -8.0000, A 0.000, B 0.000, C 0.000 }
gfCNCPoint5[27479] = {X 462.3117, Y 16.3099, Z -8.0000, A 0.000, B 0.000, C 0.000 }
gfCNCPoint5[27480] = {X 462.3113, Y 16.7691, Z -8.0000, A 0.000, B 0.000, C 0.000 }
gfCNCPoint5[27481] = {X 462.3123, Y 40.8774, Z -8.0000, A 0.000, B 0.000, C 0.000 }
gfCNCPoint5[27482] = {X 462.9561, Y 41.5664, Z -8.0000, A 0.000, B 0.000, C 0.000 }
gfCNCPoint5[27483] = {X 463.4384, Y 42.3767, Z -8.0000, A 0.000, B 0.000, C 0.000 }
gfCNCPoint5[27484] = {X 463.7369, Y 43.2713, Z -8.0000, A 0.000, B 0.000, C 0.000 }
gfCNCPoint5[27485] = {X 463.8379, Y 44.2088, Z -8.0000, A 0.000, B 0.000, C 0.000 }
gfCNCPoint5[27486] = {X 463.8379, Y 45.0000, Z -8.0000, A 0.000, B 0.000, C 0.000 }
gfCNCPoint5[27487] = {X 463.7612, Y 45.8182, Z -8.0000, A 0.000, B 0.000, C 0.000 }
gfCNCPoint5[27488] = {X 463.5336, Y 46.6079, Z -8.0000, A 0.000, B 0.000, C 0.000 }
gfCNCPoint5[27489] = {X 463.1632, Y 47.3415, Z -8.0000, A 0.000, B 0.000, C 0.000 }
gfCNCPoint5[27490] = {X 462.6627, Y 47.9934, Z -8.0000, A 0.000, B 0.000, C 0.000 }
gfCNCPoint5[27491] = {X 463.0145, Y 48.3200, Z -8.0000, A 0.000, B 0.000, C 0.000 }
gfCNCPoint5[27492] = {X 472.1884, Y 48.3200, Z -8.0000, A 0.000, B 0.000, C 0.000 }
gfCNCPoint5[27493] = {X 471.5820, Y 47.5134, Z -8.0000, A 0.000, B 0.000, C 0.000 }
gfCNCPoint5[27494] = {X 471.1544, Y 46.5992, Z -8.0000, A 0.000, B 0.000, C 0.000 }
gfCNCPoint5[27495] = {X 470.9241, Y 45.6167, Z -8.0000, A 0.000, B 0.000, C 0.000 }
gfCNCPoint5[27496] = {X 470.8947, Y 45.3090, Z -8.0000, A 0.000, B 0.000, C 0.000 }
gfCNCPoint5[27497] = {X 470.8850, Y 45.0000, Z -8.0000, A 0.000, B 0.000, C 0.000 }
gfCNCPoint5[27498] = {X 470.8850, Y 44.2089, Z -8.0000, A 0.000, B 0.000, C 0.000 }
gfCNCPoint5[27499] = {X 470.9769, Y 43.2661, Z -8.0000, A 0.000, B 0.000, C 0.000 }
gfCNCPoint5[27500] = {X 471.2492, Y 42.3588, Z -8.0000, A 0.000, B 0.000, C 0.000 }
gfCNCPoint5[27501] = {X 471.6917, Y 41.5212, Z -8.0000, A 0.000, B 0.000, C 0.000 }
gfCNCPoint5[27502] = {X 472.2877, Y 40.7849, Z -8.0000, A 0.000, B 0.000, C 0.000 }
gfCNCPoint5[27503] = {X 473.0147, Y 40.1776, Z -8.0000, A 0.000, B 0.000, C 0.000 }
gfCNCPoint5[27504] = {X 473.8453, Y 39.7222, Z -8.0000, A 0.000, B 0.000, C 0.000 }
gfCNCPoint5[27505] = {X 477.5000, Y 32.5684, Z -8.0000, A 0.000, B 0.000, C 0.000 }
gfCNCPoint5[27506] = {X 476.2820, Y 31.6589, Z -8.0000, A 0.000, B 0.000, C 0.000 }
gfCNCPoint5[27507] = {X 475.1885, Y 30.6029, Z -8.0000, A 0.000, B 0.000, C 0.000 }
gfCNCPoint5[27508] = {X 474.2371, Y 29.4172, Z -8.0000, A 0.000, B 0.000, C 0.000 }
gfCNCPoint5[27509] = {X 473.4431, Y 28.1209, Z -8.0000, A 0.000, B 0.000, C 0.000 }
gfCNCPoint5[27510] = {X 472.8192, Y 26.7347, Z -8.0000, A 0.000, B 0.000, C 0.000 }
gfCNCPoint5[27511] = {X 472.3753, Y 25.2808, Z -8.0000, A 0.000, B 0.000, C 0.000 }
gfCNCPoint5[27512] = {X 472.0514, Y 23.5415, Z -8.0000, A 0.000, B 0.000, C 0.000 }
gfCNCPoint5[27513] = {X 471.9066, Y 21.7784, Z -8.0000, A 0.000, B 0.000, C 0.000 }
gfCNCPoint5[27514] = {X 471.9425, Y 20.0096, Z -8.0000, A 0.000, B 0.000, C 0.000 }
gfCNCPoint5[27515] = {X 472.1587, Y 18.2537, Z -8.0000, A 0.000, B 0.000, C 0.000 }
gfCNCPoint5[27516] = {X 472.5530, Y 16.5291, Z -8.0000, A 0.000, B 0.000, C 0.000 }
gfCNCPoint5[27517] = {X 473.0718, Y 15.0580, Z -8.0000, A 0.000, B 0.000, C 0.000 }
gfCNCPoint5[27518] = {X 473.7713, Y 13.6637, Z -8.0000, A 0.000, B 0.000, C 0.000 }
gfCNCPoint5[27519] = {X 474.6404, Y 12.3684, Z -8.0000, A 0.000, B 0.000, C 0.000 }
gfCNCPoint5[27520] = {X 475.6653, Y 11.1924, Z -8.0000, A 0.000, B 0.000, C 0.000 }
gfCNCPoint5[27521] = {X 476.7430, Y 10.2231, Z -8.0000, A 0.000, B 0.000, C 0.000 }
gfCNCPoint5[27522] = {X 477.9264, Y 9.3862, Z -8.0000, A 0.000, B 0.000, C 0.000 }
gfCNCPoint5[27523] = {X 479.1995, Y 8.6932, Z -8.0000, A 0.000, B 0.000, C 0.000 }
gfCNCPoint5[27524] = {X 480.5447, Y 8.1536, Z -8.0000, A 0.000, B 0.000, C 0.000 }
gfCNCPoint5[27525] = {X 481.9437, Y 7.7746, Z -8.0000, A 0.000, B 0.000, C 0.000 }
gfCNCPoint5[27526] = {X 484.0948, Y 7.4393, Z -8.0000, A 0.000, B 0.000, C 0.000 }
gfCNCPoint5[27527] = {X 486.2687, Y 7.3214, Z -8.0000, A 0.000, B 0.000, C 0.000 }
gfCNCPoint5[27528] = {X 486.9707, Y 7.3092, Z -8.0000, A 0.000, B 0.000, C 0.000 }
gfCNCPoint5[27529] = {X 502.2122, Y 7.3093, Z -8.0000, A 0.000, B 0.000, C 0.000 }
gfCNCPoint5[27530] = {X 502.7438, Y 7.3134, Z -8.0000, A 0.000, B 0.000, C 0.000 }
gfCNCPoint5[27531] = {X 503.6983, Y 7.4156, Z -8.0000, A 0.000, B 0.000, C 0.000 }
gfCNCPoint5[27532] = {X 504.6140, Y 7.7033, Z -8.0000, A 0.000, B 0.000, C 0.000 }
gfCNCPoint5[27533] = {X 505.4555, Y 8.1653, Z -8.0000, A 0.000, B 0.000, C 0.000 }
gfCNCPoint5[27534] = {X 506.1897, Y 8.7836, Z -8.0000, A 0.000, B 0.000, C 0.000 }
gfCNCPoint5[27535] = {X 506.7882, Y 9.5341, Z -8.0000, A 0.000, B 0.000, C 0.000 }
gfCNCPoint5[27536] = {X 507.2277, Y 10.3875, Z -8.0000, A 0.000, B 0.000, C 0.000 }
gfCNCPoint5[27537] = {X 507.4825, Y 11.2656, Z -8.0000, A 0.000, B 0.000, C 0.000 }
gfCNCPoint5[27538] = {X 507.5685, Y 12.1759, Z -8.0000, A 0.000, B 0.000, C 0.000 }
gfCNCPoint5[27539] = {X 507.5683, Y 13.0237, Z -8.0000, A 0.000, B 0.000, C 0.000 }
gfCNCPoint5[27540] = {X 507.4609, Y 13.9969, Z -8.0000, A 0.000, B 0.000, C 0.000 }
gfCNCPoint5[27541] = {X 507.1615, Y 14.9290, Z -8.0000, A 0.000, B 0.000, C 0.000 }
gfCNCPoint5[27542] = {X 506.6820, Y 15.7827, Z -8.0000, A 0.000, B 0.000, C 0.000 }
gfCNCPoint5[27543] = {X 506.0418, Y 16.5234, Z -8.0000, A 0.000, B 0.000, C 0.000 }
gfCNCPoint5[27544] = {X 506.0423, Y 40.6639, Z -8.0000, A 0.000, B 0.000, C 0.000 }
gfCNCPoint5[27545] = {X 506.6828, Y 41.4053, Z -8.0000, A 0.000, B 0.000, C 0.000 }
gfCNCPoint5[27546] = {X 507.1623, Y 42.2597, Z -8.0000, A 0.000, B 0.000, C 0.000 }
gfCNCPoint5[27547] = {X 507.4615, Y 43.1926, Z -8.0000, A 0.000, B 0.000, C 0.000 }
gfCNCPoint5[27548] = {X 507.5683, Y 44.1665, Z -8.0000, A 0.000, B 0.000, C 0.000 }
gfCNCPoint5[27549] = {X 507.5685, Y 45.0000, Z -8.0000, A 0.000, B 0.000, C 0.000 }
gfCNCPoint5[27550] = {X 507.4747, Y 45.9520, Z -8.0000, A 0.000, B 0.000, C 0.000 }
gfCNCPoint5[27551] = {X 507.1970, Y 46.8675, Z -8.0000, A 0.000, B 0.000, C 0.000 }
gfCNCPoint5[27552] = {X 506.7461, Y 47.7112, Z -8.0000, A 0.000, B 0.000, C 0.000 }
gfCNCPoint5[27553] = {X 506.1392, Y 48.4507, Z -8.0000, A 0.000, B 0.000, C 0.000 }
gfCNCPoint5[27554] = {X 505.3997, Y 49.0576, Z -8.0000, A 0.000, B 0.000, C 0.000 }
gfCNCPoint5[27555] = {X 504.5560, Y 49.5085, Z -8.0000, A 0.000, B 0.000, C 0.000 }
gfCNCPoint5[27556] = {X 503.6405, Y 49.7862, Z -8.0000, A 0.000, B 0.000, C 0.000 }
gfCNCPoint5[27557] = {X 502.6885, Y 49.8800, Z -8.0000, A 0.000, B 0.000, C 0.000 }
gfCNCPoint5[27558] = {X 496.2450, Y 49.8800, Z -8.0000, A 0.000, B 0.000, C 0.000 }
gfCNCPoint5[27559] = {X 495.2220, Y 49.7716, Z -8.0000, A 0.000, B 0.000, C 0.000 }
gfCNCPoint5[27560] = {X 494.2445, Y 49.4511, Z -8.0000, A 0.000, B 0.000, C 0.000 }
gfCNCPoint5[27561] = {X 493.3559, Y 48.9328, Z -8.0000, A 0.000, B 0.000, C 0.000 }
gfCNCPoint5[27562] = {X 492.5956, Y 48.2398, Z -8.0000, A 0.000, B 0.000, C 0.000 }
gfCNCPoint5[27563] = {X 491.9976, Y 47.4028, Z -8.0000, A 0.000, B 0.000, C 0.000 }
gfCNCPoint5[27564] = {X 491.5882, Y 46.4590, Z -8.0000, A 0.000, B 0.000, C 0.000 }
gfCNCPoint5[27565] = {X 491.4241, Y 45.7570, Z -8.0000, A 0.000, B 0.000, C 0.000 }
gfCNCPoint5[27566] = {X 491.3652, Y 45.0385, Z -8.0000, A 0.000, B 0.000, C 0.000 }
gfCNCPoint5[27567] = {X 491.3655, Y 44.1417, Z -8.0000, A 0.000, B 0.000, C 0.000 }
gfCNCPoint5[27568] = {X 491.4758, Y 43.1751, Z -8.0000, A 0.000, B 0.000, C 0.000 }
gfCNCPoint5[27569] = {X 491.7755, Y 42.2497, Z -8.0000, A 0.000, B 0.000, C 0.000 }
gfCNCPoint5[27570] = {X 492.2530, Y 41.4021, Z -8.0000, A 0.000, B 0.000, C 0.000 }
